C05446=1006.982,330.511,340.600,169.675,53.827,160.488
C05447=1006.976,330.263,340.633,169.667,53.832,160.487
C05448=1006.972,330.016,340.666,169.659,53.837,160.487
C05449=1006.965,329.768,340.699,169.651,53.842,160.486
C05450=1006.960,329.520,340.733,169.643,53.848,160.486
C05451=1006.954,329.273,340.766,169.635,53.853,160.485
C05452=1006.948,329.025,340.799,169.629,53.858,160.485
C05453=1006.942,328.777,340.832,169.620,53.863,160.484
C05454=1006.937,328.530,340.864,169.613,53.869,160.484
C05455=1006.931,328.282,340.897,169.605,53.874,160.483
C05456=1006.926,328.034,340.930,169.597,53.879,160.483
C05457=1006.919,327.786,340.963,169.589,53.885,160.483
C05458=1006.915,327.538,340.995,169.582,53.890,160.482
C05459=1006.909,327.290,341.029,169.575,53.895,160.482
C05460=1006.903,327.043,341.061,169.567,53.900,160.481
C05461=1006.897,326.795,341.095,169.559,53.906,160.481
C05462=1006.893,326.547,341.127,169.552,53.911,160.481
C05463=1006.886,326.300,341.160,169.544,53.916,160.480
C05464=1006.881,326.051,341.192,169.537,53.922,160.480
C05465=1006.876,325.804,341.225,169.529,53.927,160.480
C05466=1006.870,325.556,341.258,169.521,53.932,160.479
C05467=1006.865,325.308,341.290,169.514,53.938,160.479
C05468=1006.859,325.061,341.323,169.507,53.943,160.478
C05469=1006.852,324.704,341.370,169.495,53.951,160.478
C05470=1006.844,324.349,341.417,169.485,53.959,160.477
C05471=1006.835,323.993,341.462,169.474,53.967,160.477
C05472=1006.827,323.638,341.509,169.464,53.974,160.476
C05473=1006.822,323.391,341.540,169.456,53.980,160.476
C05474=1006.816,323.142,341.572,169.449,53.985,160.476
C05475=1006.810,322.895,341.604,169.441,53.990,160.475
C05476=1006.805,322.646,341.637,169.434,53.996,160.475
C05477=1006.800,322.399,341.668,169.426,54.001,160.474
C05478=1006.794,322.151,341.700,169.419,54.007,160.474
C05479=1006.788,321.903,341.732,169.411,54.013,160.474
C05480=1006.782,321.655,341.764,169.404,54.018,160.474
C05481=1006.778,321.407,341.796,169.397,54.024,160.473
C05482=1006.772,321.159,341.828,169.389,54.029,160.473
C05483=1006.766,320.911,341.860,169.382,54.035,160.473
C05484=1006.760,320.663,341.892,169.375,54.040,160.472
C05485=1006.755,320.416,341.924,169.367,54.046,160.472
C05486=1006.749,320.168,341.955,169.360,54.051,160.472
C05487=1006.744,319.920,341.988,169.353,54.057,160.471
C05488=1006.739,319.672,342.020,169.345,54.062,160.471
C05489=1006.733,319.424,342.051,169.338,54.068,160.471
C05490=1006.727,319.176,342.083,169.330,54.074,160.470
C05491=1006.722,318.928,342.114,169.324,54.079,160.470
C05492=1006.717,318.681,342.146,169.316,54.085,160.470
C05493=1006.712,318.432,342.179,169.308,54.090,160.469
C05494=1006.706,318.185,342.210,169.302,54.096,160.469
C05495=1006.701,317.937,342.242,169.294,54.101,160.469
C05496=1006.696,317.689,342.273,169.287,54.108,160.469
C05497=1006.690,317.441,342.305,169.280,54.113,160.468
C05498=1006.685,317.193,342.337,169.273,54.118,160.468
C05499=1006.680,316.945,342.368,169.265,54.124,160.468
C05500=1006.675,316.697,342.400,169.258,54.129,160.467
C05501=1006.669,316.450,342.431,169.251,54.135,160.467
C05502=1006.664,316.202,342.462,169.244,54.141,160.467
C05503=1006.658,315.953,342.494,169.237,54.147,160.467
C05504=1006.654,315.705,342.526,169.229,54.152,160.466
C05505=1006.649,315.457,342.558,169.223,54.158,160.466
C05506=1006.643,315.209,342.589,169.215,54.163,160.466
C05507=1006.638,314.962,342.620,169.208,54.170,160.466
C05508=1006.633,314.714,342.652,169.201,54.175,160.465
C05509=1006.628,314.466,342.683,169.194,54.181,160.465
C05510=1006.623,314.218,342.714,169.187,54.187,160.465
C05511=1006.618,313.970,342.746,169.180,54.192,160.465
C05512=1006.613,313.722,342.777,169.172,54.198,160.464
C05513=1006.607,313.475,342.809,169.166,54.204,160.464
C05514=1006.602,313.226,342.840,169.159,54.210,160.464
C05515=1006.598,312.979,342.872,169.152,54.215,160.464
C05516=1006.593,312.730,342.903,169.145,54.221,160.464
C05517=1006.588,312.482,342.934,169.137,54.227,160.463
C05518=1006.582,312.235,342.965,169.130,54.232,160.463
C05519=1006.577,311.987,342.996,169.123,54.238,160.463
C05520=1006.572,311.739,343.027,169.117,54.244,160.463
C05521=1006.568,311.490,343.059,169.110,54.250,160.462
C05522=1006.562,311.243,343.090,169.102,54.256,160.462
C05523=1006.557,310.994,343.121,169.095,54.261,160.462
C05524=1006.553,310.747,343.152,169.088,54.267,160.462
C05525=1006.548,310.499,343.183,169.082,54.273,160.461
C05526=1006.543,310.251,343.214,169.074,54.279,160.461
C05527=1006.538,310.003,343.246,169.068,54.284,160.461
C05528=1006.533,309.755,343.277,169.061,54.291,160.461
C05529=1006.526,309.405,343.321,169.051,54.299,160.461
C05530=1006.519,309.055,343.365,169.041,54.307,160.460
C05531=1006.512,308.706,343.408,169.032,54.316,160.460
C05532=1006.505,308.356,343.451,169.022,54.324,160.460
C05533=1006.501,308.107,343.483,169.015,54.329,160.460
C05534=1006.496,307.860,343.513,169.008,54.336,160.459
C05535=1006.491,307.612,343.544,169.000,54.341,160.459
C05536=1006.485,307.364,343.574,168.994,54.347,160.459
C05537=1006.481,307.116,343.604,168.987,54.354,160.459
C05538=1006.475,306.868,343.634,168.981,54.359,160.459
C05539=1006.470,306.620,343.665,168.973,54.365,160.458
C05540=1006.465,306.373,343.694,168.967,54.371,160.458
C05541=1006.460,306.124,343.725,168.960,54.377,160.458
C05542=1006.454,305.876,343.755,168.954,54.383,160.458
C05543=1006.449,305.628,343.786,168.946,54.389,160.458
C05544=1006.444,305.380,343.815,168.939,54.396,160.458
C05545=1006.440,305.122,343.847,168.933,54.401,160.458
C05546=1006.434,304.865,343.878,168.926,54.407,160.457
C05547=1006.429,304.606,343.910,168.918,54.414,160.457
C05548=1006.423,304.348,343.941,168.911,54.420,160.457
C05549=1006.180,304.930,343.505,168.907,54.441,160.461
C05550=1006.187,305.298,343.459,168.917,54.432,160.461
C05551=1006.194,305.666,343.415,168.927,54.424,160.461
C05552=1006.203,306.035,343.370,168.937,54.414,160.462
C05553=1006.210,306.403,343.325,168.948,54.405,160.462
C05554=1006.215,306.650,343.295,168.954,54.399,160.462
C05555=1006.220,306.899,343.265,168.962,54.394,160.462
C05556=1006.225,307.147,343.235,168.968,54.388,160.462
C05557=1006.229,307.395,343.205,168.975,54.381,160.463
C05558=1006.235,307.643,343.175,168.982,54.376,160.463
C05559=1006.240,307.891,343.144,168.989,54.370,160.463
C05560=1006.245,308.138,343.113,168.995,54.364,160.463
C05561=1006.250,308.386,343.082,169.003,54.358,160.463
C05562=1006.257,308.739,343.039,169.012,54.350,160.464
C05563=1006.264,309.090,342.995,169.022,54.342,160.464
C05564=1006.270,309.442,342.950,169.032,54.334,160.464
C05565=1006.277,309.795,342.907,169.042,54.326,160.465
C05566=1006.282,310.043,342.876,169.049,54.319,160.465
C05567=1006.287,310.291,342.845,169.056,54.314,160.465
C05568=1006.293,310.539,342.813,169.063,54.308,160.466
C05569=1006.296,310.786,342.782,169.069,54.302,160.465
C05570=1006.301,311.035,342.751,169.077,54.297,160.466
C05571=1006.306,311.283,342.720,169.083,54.291,160.466
C05572=1006.312,311.531,342.689,169.091,54.285,160.466
C05573=1006.317,311.779,342.658,169.097,54.280,160.467
C05574=1006.321,312.027,342.626,169.104,54.273,160.467
C05575=1006.326,312.274,342.596,169.111,54.268,160.467
C05576=1006.331,312.522,342.565,169.119,54.262,160.467
C05577=1006.336,312.770,342.533,169.125,54.256,160.467
C05578=1006.341,313.018,342.502,169.133,54.251,160.468
C05579=1006.346,313.266,342.471,169.140,54.245,160.468
C05580=1006.351,313.514,342.439,169.147,54.240,160.468
C05581=1006.356,313.762,342.408,169.154,54.233,160.468
C05582=1006.361,314.010,342.377,169.161,54.228,160.469
C05583=1006.367,314.258,342.345,169.168,54.222,160.469
C05584=1006.372,314.506,342.314,169.175,54.217,160.469
C05585=1006.377,314.753,342.283,169.182,54.211,160.469
C05586=1006.381,315.002,342.251,169.190,54.205,160.470
C05587=1006.387,315.249,342.219,169.196,54.200,160.470
C05588=1006.392,315.497,342.188,169.204,54.194,160.470
C05589=1006.397,315.745,342.157,169.210,54.189,160.471
C05590=1006.402,315.993,342.126,169.218,54.183,160.471
C05591=1006.408,316.242,342.093,169.225,54.177,160.471
C05592=1006.413,316.490,342.062,169.232,54.172,160.471
C05593=1006.418,316.737,342.031,169.239,54.166,160.472
C05594=1006.423,316.985,342.000,169.247,54.160,160.472
C05595=1006.428,317.233,341.968,169.254,54.155,160.472
C05596=1006.434,317.480,341.936,169.261,54.149,160.473
C05597=1006.439,317.730,341.904,169.268,54.144,160.473
C05598=1006.444,317.977,341.873,169.276,54.138,160.473
C05599=1006.450,318.225,341.841,169.283,54.133,160.474
C05600=1006.455,318.473,341.810,169.290,54.127,160.474
C05601=1006.460,318.720,341.779,169.298,54.122,160.474
C05602=1006.466,318.968,341.747,169.305,54.116,160.475
C05603=1006.471,319.216,341.714,169.312,54.111,160.475
C05604=1006.476,319.464,341.683,169.319,54.105,160.475
C05605=1006.482,319.713,341.651,169.327,54.099,160.476
C05606=1006.487,319.960,341.620,169.334,54.094,160.476
C05607=1006.493,320.208,341.588,169.341,54.088,160.476
C05608=1006.498,320.456,341.555,169.349,54.083,160.477
C05609=1006.503,320.704,341.524,169.356,54.078,160.477
C05610=1006.509,320.951,341.492,169.363,54.072,160.477
C05611=1006.515,321.199,341.460,169.371,54.066,160.478
C05612=1006.520,321.447,341.428,169.378,54.061,160.478
C05613=1006.526,321.695,341.396,169.385,54.055,160.478
C05614=1006.531,321.943,341.364,169.393,54.050,160.478
C05615=1006.536,322.190,341.332,169.401,54.045,160.479
C05616=1006.542,322.439,341.300,169.407,54.039,160.479
C05617=1006.547,322.686,341.269,169.415,54.034,160.480
C05618=1006.553,322.934,341.237,169.423,54.028,160.480
C05619=1006.558,323.182,341.204,169.430,54.022,160.480
C05620=1006.564,323.430,341.172,169.437,54.017,160.481
C05621=1006.569,323.678,341.141,169.445,54.012,160.481
C05622=1006.578,324.036,341.095,169.456,54.004,160.482
C05623=1006.586,324.394,341.048,169.466,53.997,160.482
C05624=1006.594,324.752,341.002,169.478,53.989,160.483
C05625=1006.602,325.110,340.954,169.489,53.981,160.483
C05626=1006.607,325.358,340.922,169.495,53.976,160.484
C05627=1006.613,325.605,340.889,169.503,53.971,160.484
C05628=1006.618,325.854,340.857,169.511,53.965,160.485
C05629=1006.623,326.101,340.824,169.519,53.959,160.485
C05630=1006.629,326.348,340.791,169.526,53.955,160.485
C05631=1006.635,326.597,340.758,169.533,53.949,160.486
C05632=1006.639,326.844,340.725,169.542,53.944,160.486
C05633=1006.645,327.092,340.693,169.549,53.938,160.487
C05634=1006.651,327.340,340.660,169.556,53.933,160.487
C05635=1006.657,327.587,340.628,169.564,53.928,160.487
C05636=1006.662,327.836,340.595,169.572,53.923,160.488
C05637=1006.668,328.084,340.562,169.580,53.918,160.488
C05638=1006.674,328.331,340.529,169.587,53.912,160.489
C05639=1006.679,328.578,340.496,169.594,53.907,160.489
C05640=1006.684,328.827,340.463,169.602,53.902,160.489
C05641=1006.690,329.075,340.430,169.610,53.897,160.490
C05642=1006.696,329.322,340.397,169.618,53.891,160.490
C05643=1006.701,329.570,340.364,169.626,53.886,160.491
C05644=1006.707,329.817,340.331,169.633,53.882,160.491
C05645=1006.713,330.065,340.298,169.641,53.876,160.492
C05646=1006.719,330.313,340.265,169.649,53.871,160.492
C05647=1006.725,330.561,340.232,169.656,53.865,160.493
C05648=1006.730,330.809,340.199,169.664,53.860,160.493
C05649=1006.736,331.056,340.166,169.672,53.856,160.494
C05650=1006.741,331.303,340.133,169.679,53.850,160.494
C05651=1006.747,331.551,340.100,169.687,53.845,160.495
C05652=1006.752,331.799,340.066,169.695,53.840,160.495
C05653=1006.758,332.047,340.033,169.703,53.835,160.496
C05654=1006.764,332.295,340.000,169.711,53.830,160.496
C05655=1006.769,332.542,339.966,169.718,53.825,160.497
C05656=1006.775,332.790,339.932,169.726,53.820,160.497
C05657=1006.780,333.038,339.899,169.734,53.815,160.498
C05658=1006.787,333.286,339.866,169.742,53.809,160.498
C05659=1006.793,333.533,339.832,169.750,53.804,160.499
C05660=1006.798,333.781,339.799,169.758,53.800,160.499
C05661=1006.804,334.029,339.765,169.766,53.795,160.500
C05662=1006.810,334.276,339.731,169.774,53.790,160.500
C05663=1006.815,334.524,339.698,169.782,53.785,160.501
C05664=1006.821,334.771,339.664,169.789,53.779,160.501
C05665=1006.827,335.019,339.631,169.797,53.774,160.502
C05666=1006.833,335.268,339.597,169.805,53.769,160.502
C05667=1006.839,335.515,339.563,169.813,53.765,160.503
C05668=1006.845,335.763,339.530,169.822,53.760,160.503
C05669=1006.851,336.010,339.496,169.830,53.755,160.504
C05670=1006.857,336.257,339.462,169.838,53.750,160.504
C05671=1006.862,336.505,339.429,169.846,53.745,160.505
C05672=1006.869,336.753,339.394,169.854,53.740,160.506
C05673=1006.874,337.001,339.361,169.862,53.735,160.506
C05674=1006.880,337.248,339.327,169.870,53.730,160.507
C05675=1006.886,337.496,339.293,169.877,53.725,160.507
C05676=1006.892,337.744,339.258,169.885,53.720,160.508
C05677=1006.898,337.991,339.225,169.893,53.715,160.508
C05678=1006.904,338.239,339.191,169.902,53.710,160.509
C05679=1006.910,338.486,339.157,169.910,53.706,160.510
C05680=1006.916,338.734,339.123,169.918,53.701,160.510
C05681=1006.921,338.982,339.088,169.926,53.696,160.511
C05682=1006.929,339.306,339.043,169.937,53.689,160.511
C05683=1006.937,339.630,338.999,169.948,53.683,160.512
C05684=1006.945,339.955,338.953,169.958,53.677,160.513
C05685=1006.953,340.279,338.909,169.969,53.671,160.514
C05686=1006.959,340.527,338.874,169.977,53.666,160.515
C05687=1006.964,340.774,338.839,169.985,53.661,160.515
C05688=1006.971,341.022,338.805,169.994,53.656,160.516
C05689=1006.977,341.270,338.771,170.002,53.651,160.516
C05690=1006.983,341.518,338.737,170.010,53.647,160.517
C05691=1006.989,341.765,338.703,170.018,53.642,160.518
C05692=1006.995,342.013,338.667,170.026,53.637,160.518
C05693=1007.001,342.260,338.633,170.035,53.633,160.519
C05694=1007.007,342.508,338.598,170.043,53.628,160.519
C05695=1007.013,342.755,338.564,170.052,53.624,160.520
C05696=1007.020,343.003,338.529,170.060,53.619,160.521
C05697=1007.025,343.250,338.494,170.068,53.614,160.521
C05698=1007.032,343.498,338.459,170.076,53.610,160.522
C05699=1007.038,343.745,338.425,170.085,53.605,160.523
C05700=1007.044,343.993,338.391,170.093,53.600,160.523
C05701=1007.050,344.240,338.355,170.102,53.595,160.524
C05702=1006.736,342.085,338.297,170.011,53.676,160.524
C05703=1006.730,341.839,338.332,170.002,53.680,160.523
C05704=1006.724,341.591,338.366,169.994,53.685,160.523
C05705=1006.718,341.343,338.401,169.986,53.690,160.522
C05706=1006.713,341.096,338.435,169.978,53.695,160.521
C05707=1006.706,340.848,338.470,169.970,53.700,160.521
C05708=1006.700,340.600,338.504,169.961,53.704,160.520
C05709=1006.694,340.353,338.538,169.953,53.709,160.520
C05710=1006.688,340.105,338.572,169.945,53.714,160.519
C05711=1006.682,339.837,338.609,169.936,53.719,160.518
C05712=1006.676,339.568,338.647,169.927,53.725,160.518
C05713=1006.669,339.300,338.685,169.918,53.729,160.517
C05714=1006.663,339.031,338.721,169.909,53.734,160.516
C05715=1006.657,338.784,338.755,169.901,53.739,160.516
C05716=1006.651,338.536,338.789,169.893,53.744,160.515
C05717=1006.645,338.289,338.823,169.885,53.749,160.515
C05718=1006.639,338.041,338.857,169.876,53.754,160.514
C05719=1006.633,337.794,338.891,169.868,53.758,160.513
C05720=1006.628,337.545,338.926,169.860,53.763,160.513
C05721=1006.622,337.298,338.960,169.853,53.768,160.512
C05722=1006.616,337.050,338.994,169.845,53.773,160.512
C05723=1006.610,336.803,339.027,169.837,53.778,160.511
C05724=1006.604,336.556,339.061,169.828,53.783,160.510
C05725=1006.597,336.307,339.094,169.820,53.788,160.510
C05726=1006.592,336.060,339.128,169.812,53.793,160.509
C05727=1006.586,335.812,339.162,169.804,53.798,160.509
C05728=1006.580,335.565,339.196,169.796,53.803,160.508
C05729=1006.575,335.317,339.229,169.788,53.808,160.508
C05730=1006.569,335.069,339.263,169.780,53.813,160.507
C05731=1006.563,334.821,339.297,169.773,53.817,160.507
C05732=1006.557,334.574,339.331,169.765,53.822,160.506
C05733=1006.551,334.327,339.363,169.757,53.827,160.505
C05734=1006.546,334.079,339.397,169.748,53.832,160.505
C05735=1006.540,333.831,339.431,169.740,53.837,160.504
C05736=1006.534,333.583,339.464,169.733,53.843,160.504
C05737=1006.529,333.336,339.497,169.725,53.848,160.503
C05738=1006.523,333.088,339.531,169.716,53.853,160.503
C05739=1006.517,332.840,339.565,169.709,53.857,160.502
C05740=1006.512,332.592,339.598,169.701,53.862,160.502
C05741=1006.506,332.345,339.631,169.693,53.867,160.501
C05742=1006.500,332.097,339.665,169.686,53.873,160.501
C05743=1006.494,331.849,339.698,169.677,53.878,160.500
C05744=1006.489,331.601,339.731,169.670,53.882,160.500
C05745=1006.483,331.354,339.765,169.662,53.887,160.499
C05746=1006.477,331.106,339.798,169.654,53.892,160.499
C05747=1006.472,330.858,339.832,169.646,53.898,160.498
C05748=1006.467,330.611,339.865,169.638,53.903,160.498
C05749=1006.460,330.363,339.897,169.630,53.908,160.497
C05750=1006.455,330.115,339.930,169.624,53.913,160.497
C05751=1006.449,329.867,339.963,169.616,53.918,160.496
C05752=1006.443,329.619,339.996,169.607,53.923,160.496
C05753=1006.438,329.372,340.029,169.600,53.929,160.495
C05754=1006.432,329.124,340.062,169.592,53.934,160.495
C05755=1006.427,328.876,340.094,169.585,53.939,160.495
C05756=1006.421,328.628,340.128,169.577,53.944,160.494
C05757=1006.416,328.381,340.160,169.569,53.949,160.493
C05758=1006.410,328.133,340.193,169.561,53.954,160.493
C05759=1006.405,327.885,340.226,169.554,53.959,160.493
C05760=1006.399,327.638,340.258,169.547,53.965,160.492
C05761=1006.394,327.390,340.292,169.538,53.970,160.492
C05762=1006.388,327.142,340.324,169.531,53.975,160.491
C05763=1006.383,326.894,340.357,169.524,53.980,160.491
C05764=1006.377,326.646,340.389,169.516,53.986,160.491
C05765=1006.371,326.398,340.422,169.508,53.991,160.490
C05766=1006.366,326.151,340.454,169.500,53.996,160.490
C05767=1006.361,325.903,340.488,169.493,54.001,160.489
C05768=1006.355,325.656,340.520,169.486,54.006,160.489
C05769=1006.350,325.407,340.553,169.478,54.012,160.488
C05770=1006.345,325.159,340.585,169.470,54.017,160.488
C05771=1006.337,324.799,340.633,169.460,54.025,160.487
C05772=1006.329,324.439,340.680,169.448,54.033,160.487
C05773=1006.321,324.078,340.726,169.437,54.041,160.486
C05774=1006.312,323.719,340.772,169.427,54.048,160.486
C05775=1006.307,323.470,340.805,169.419,54.053,160.485
C05776=1006.302,323.222,340.837,169.411,54.059,160.485
C05777=1006.296,322.974,340.869,169.405,54.064,160.485
C05778=1006.290,322.727,340.900,169.397,54.070,160.484
C05779=1006.284,322.479,340.932,169.389,54.075,160.484
C05780=1006.280,322.231,340.965,169.381,54.080,160.483
C05781=1006.274,321.983,340.996,169.375,54.086,160.483
C05782=1006.268,321.735,341.028,169.367,54.091,160.483
C05783=1006.263,321.487,341.060,169.360,54.097,160.482
C05784=1006.257,321.239,341.092,169.352,54.102,160.482
C05785=1006.252,320.992,341.124,169.345,54.107,160.481
C05786=1006.247,320.744,341.156,169.337,54.113,160.481
C05787=1006.241,320.496,341.188,169.331,54.118,160.481
C05788=1006.235,320.248,341.220,169.323,54.124,160.480
C05789=1006.230,320.000,341.250,169.315,54.129,160.480
C05790=1006.224,319.752,341.282,169.309,54.135,160.480
C05791=1006.219,319.504,341.314,169.301,54.140,160.479
C05792=1006.214,319.257,341.346,169.293,54.145,160.479
C05793=1006.209,319.009,341.378,169.286,54.151,160.479
C05794=1006.203,318.760,341.409,169.279,54.156,160.478
C05795=1006.198,318.513,341.441,169.271,54.162,160.478
C05796=1006.193,318.265,341.473,169.264,54.167,160.478
C05797=1006.188,318.017,341.504,169.257,54.173,160.477
C05798=1006.183,317.769,341.536,169.250,54.178,160.477
C05799=1006.177,317.521,341.568,169.242,54.184,160.477
C05800=1006.172,317.273,341.599,169.235,54.190,160.476
C05801=1006.166,317.025,341.631,169.228,54.195,160.476
C05802=1006.161,316.777,341.661,169.221,54.201,160.476
C05803=1006.157,316.529,341.694,169.214,54.206,160.475
C05804=1006.152,316.281,341.725,169.206,54.212,160.475
C05805=1006.146,316.034,341.756,169.199,54.218,160.475
C05806=1006.141,315.786,341.787,169.193,54.223,160.475
C05807=1006.136,315.538,341.819,169.185,54.229,160.474
C05808=1006.131,315.290,341.850,169.178,54.234,160.474
C05809=1006.126,315.042,341.882,169.171,54.240,160.474
C05810=1006.121,314.794,341.913,169.163,54.246,160.473
C05811=1006.116,314.546,341.945,169.156,54.251,160.473
C05812=1006.110,314.298,341.976,169.149,54.257,160.473
C05813=1006.105,314.050,342.007,169.143,54.262,160.473
C05814=1006.101,313.802,342.039,169.135,54.268,160.472
C05815=1006.096,313.554,342.070,169.128,54.273,160.472
C05816=1006.091,313.306,342.101,169.121,54.279,160.472
C05817=1006.085,313.059,342.132,169.114,54.284,160.471
C05818=1006.080,312.810,342.163,169.107,54.290,160.471
C05819=1006.075,312.562,342.194,169.100,54.296,160.471
C05820=1006.071,312.314,342.226,169.093,54.302,160.471
C05821=1006.065,312.066,342.258,169.086,54.307,160.470
C05822=1006.061,311.819,342.288,169.079,54.313,160.470
C05823=1006.056,311.571,342.319,169.071,54.319,160.470
C05824=1006.051,311.323,342.350,169.065,54.324,160.470
C05825=1006.046,311.074,342.382,169.057,54.330,160.469
C05826=1006.041,310.826,342.413,169.051,54.336,160.469
C05827=1006.036,310.578,342.443,169.043,54.342,160.469
C05828=1006.031,310.331,342.475,169.037,54.347,160.469
C05829=1006.026,310.083,342.506,169.030,54.353,160.468
C05830=1006.021,309.835,342.537,169.023,54.359,160.468
C05831=1006.015,309.480,342.581,169.013,54.367,160.468
C05832=1006.008,309.126,342.625,169.004,54.375,160.468
C05833=1006.002,308.772,342.669,168.993,54.383,160.467
C05834=1005.994,308.417,342.713,168.984,54.391,160.467
C05835=1005.989,308.169,342.744,168.977,54.398,160.467
C05836=1005.985,307.922,342.775,168.970,54.403,160.466
C05837=1005.980,307.673,342.806,168.963,54.409,160.466
C05838=1005.975,307.426,342.835,168.956,54.415,160.466
C05839=1005.970,307.184,342.865,168.949,54.421,160.466
C05840=1005.965,306.942,342.895,168.942,54.426,160.466
C05841=1005.960,306.700,342.924,168.936,54.432,160.465
C05842=1005.955,306.459,342.953,168.930,54.438,160.465
C05843=1005.950,306.217,342.983,168.922,54.443,160.465
C05844=1005.945,305.976,343.012,168.916,54.449,160.465
C05845=1005.941,305.734,343.041,168.909,54.455,160.465
C05846=1005.935,305.492,343.070,168.902,54.461,160.464
C05847=1005.691,306.038,342.638,168.898,54.480,160.468
C05848=1005.698,306.392,342.595,168.908,54.471,160.468
C05849=1005.705,306.747,342.553,168.918,54.463,160.468
C05850=1005.713,307.102,342.509,168.928,54.454,160.469
C05851=1005.719,307.456,342.466,168.937,54.446,160.469
C05852=1005.725,307.704,342.436,168.944,54.441,160.469
C05853=1005.730,307.952,342.405,168.951,54.434,160.469
C05854=1005.735,308.200,342.374,168.958,54.429,160.470
C05855=1005.739,308.448,342.344,168.965,54.423,160.470
C05856=1005.746,308.805,342.300,168.975,54.415,160.470
C05857=1005.753,309.162,342.256,168.985,54.407,160.471
C05858=1005.760,309.517,342.211,168.994,54.398,160.471
C05859=1005.766,309.874,342.166,169.004,54.390,160.471
C05860=1005.772,310.122,342.135,169.012,54.384,160.472
C05861=1005.777,310.370,342.104,169.018,54.379,160.472
C05862=1005.781,310.619,342.073,169.026,54.373,160.472
C05863=1005.785,310.866,342.042,169.032,54.367,160.472
C05864=1005.790,311.114,342.011,169.040,54.362,160.473
C05865=1005.796,311.362,341.980,169.046,54.356,160.473
C05866=1005.801,311.611,341.949,169.053,54.351,160.473
C05867=1005.805,311.859,341.918,169.061,54.345,160.474
C05868=1005.809,312.106,341.887,169.067,54.339,160.474
C05869=1005.815,312.354,341.856,169.074,54.334,160.474
C05870=1005.820,312.602,341.825,169.081,54.328,160.474
C05871=1005.825,312.850,341.794,169.089,54.323,160.475
C05872=1005.830,313.098,341.763,169.095,54.317,160.475
C05873=1005.834,313.347,341.731,169.103,54.312,160.475
C05874=1005.839,313.594,341.700,169.109,54.306,160.475
C05875=1005.844,313.842,341.669,169.117,54.300,160.476
C05876=1005.849,314.090,341.638,169.124,54.294,160.476
C05877=1005.855,314.337,341.606,169.131,54.289,160.476
C05878=1005.860,314.586,341.575,169.139,54.283,160.477
C05879=1005.864,314.834,341.544,169.145,54.278,160.477
C05880=1005.870,315.081,341.512,169.153,54.272,160.477
C05881=1005.875,315.330,341.481,169.160,54.267,160.478
C05882=1005.880,315.578,341.450,169.167,54.262,160.478
C05883=1005.885,315.825,341.419,169.174,54.256,160.478
C05884=1005.889,316.074,341.387,169.181,54.251,160.479
C05885=1005.895,316.321,341.356,169.188,54.245,160.479
C05886=1005.900,316.569,341.325,169.196,54.240,160.479
C05887=1005.905,316.817,341.293,169.203,54.234,160.480
C05888=1005.911,317.066,341.262,169.210,54.229,160.480
C05889=1005.916,317.313,341.230,169.218,54.223,160.480
C05890=1005.921,317.562,341.198,169.224,54.218,160.480
C05891=1005.926,317.809,341.167,169.232,54.212,160.481
C05892=1005.931,318.057,341.135,169.239,54.206,160.481
C05893=1005.937,318.305,341.104,169.246,54.201,160.481
C05894=1005.942,318.552,341.072,169.254,54.195,160.482
C05895=1005.947,318.801,341.040,169.260,54.190,160.482
C05896=1005.952,319.049,341.009,169.268,54.184,160.482
C05897=1005.958,319.296,340.977,169.276,54.179,160.483
C05898=1005.963,319.544,340.946,169.283,54.174,160.483
C05899=1005.969,319.793,340.914,169.290,54.168,160.484
C05900=1005.974,320.040,340.883,169.297,54.163,160.484
C05901=1005.979,320.288,340.850,169.305,54.157,160.484
C05902=1005.984,320.536,340.819,169.312,54.152,160.485
C05903=1005.990,320.785,340.787,169.319,54.147,160.485
C05904=1005.995,321.032,340.756,169.327,54.141,160.485
C05905=1006.001,321.280,340.724,169.335,54.136,160.486
C05906=1006.006,321.528,340.691,169.341,54.131,160.486
C05907=1006.011,321.776,340.660,169.349,54.126,160.487
C05908=1006.017,322.023,340.628,169.357,54.120,160.487
C05909=1006.023,322.271,340.596,169.364,54.115,160.487
C05910=1006.028,322.519,340.564,169.371,54.109,160.488
C05911=1006.034,322.767,340.532,169.379,54.104,160.488
C05912=1006.039,323.015,340.500,169.386,54.099,160.489
C05913=1006.044,323.262,340.468,169.394,54.093,160.489
C05914=1006.050,323.511,340.436,169.402,54.088,160.489
C05915=1006.055,323.758,340.405,169.409,54.082,160.490
C05916=1006.064,324.121,340.359,169.419,54.075,160.490
C05917=1006.072,324.484,340.311,169.431,54.067,160.491
C05918=1006.080,324.846,340.263,169.442,54.059,160.492
C05919=1006.087,325.209,340.216,169.452,54.052,160.492
C05920=1006.093,325.457,340.184,169.460,54.046,160.493
C05921=1006.098,325.705,340.151,169.468,54.041,160.493
C05922=1006.104,325.953,340.118,169.476,54.036,160.494
C05923=1006.109,326.200,340.086,169.483,54.031,160.494
C05924=1006.114,326.448,340.053,169.491,54.025,160.494
C05925=1006.119,326.696,340.021,169.499,54.020,160.495
C05926=1006.125,326.943,339.988,169.505,54.015,160.495
C05927=1006.131,327.192,339.955,169.513,54.010,160.496
C05928=1006.136,327.439,339.923,169.521,54.005,160.496
C05929=1006.142,327.687,339.890,169.529,54.000,160.497
C05930=1006.147,327.935,339.857,169.536,53.995,160.497
C05931=1006.153,328.182,339.825,169.544,53.989,160.498
C05932=1006.158,328.431,339.792,169.552,53.984,160.498
C05933=1006.164,328.679,339.759,169.560,53.979,160.498
C05934=1006.169,328.925,339.726,169.567,53.974,160.499
C05935=1006.175,329.173,339.693,169.575,53.969,160.500
C05936=1006.180,329.422,339.660,169.582,53.963,160.500
C05937=1006.186,329.670,339.628,169.591,53.958,160.500
C05938=1006.191,329.917,339.595,169.598,53.954,160.501
C05939=1006.198,330.164,339.562,169.606,53.949,160.502
C05940=1006.203,330.412,339.528,169.613,53.943,160.502
C05941=1006.208,330.661,339.496,169.622,53.938,160.502
C05942=1006.214,330.908,339.463,169.630,53.933,160.503
C05943=1006.220,331.156,339.430,169.637,53.929,160.504
C05944=1006.225,331.403,339.397,169.644,53.923,160.504
C05945=1006.231,331.651,339.363,169.652,53.918,160.504
C05946=1006.237,331.899,339.329,169.661,53.913,160.505
C05947=1006.242,332.147,339.296,169.669,53.908,160.506
C05948=1006.248,332.394,339.263,169.676,53.904,160.506
C05949=1006.253,332.642,339.230,169.684,53.899,160.507
C05950=1006.258,332.890,339.196,169.691,53.893,160.507
C05951=1006.265,333.137,339.164,169.700,53.888,160.508
C05952=1006.270,333.385,339.130,169.708,53.883,160.508
C05953=1006.276,333.632,339.096,169.715,53.878,160.509
C05954=1006.282,333.880,339.063,169.723,53.873,160.509
C05955=1006.287,334.128,339.030,169.731,53.868,160.510
C05956=1006.293,334.375,338.996,169.739,53.863,160.510
C05957=1006.299,334.623,338.962,169.747,53.858,160.511
C05958=1006.304,334.871,338.929,169.755,53.854,160.512
C05959=1006.310,335.119,338.895,169.763,53.849,160.512
C05960=1006.316,335.366,338.862,169.771,53.844,160.513
C05961=1006.322,335.614,338.829,169.779,53.839,160.513
C05962=1006.328,335.862,338.794,169.787,53.834,160.514
C05963=1006.334,336.110,338.761,169.795,53.829,160.514
C05964=1006.340,336.357,338.727,169.803,53.824,160.515
C05965=1006.345,336.605,338.694,169.811,53.819,160.515
C05966=1006.351,336.852,338.660,169.819,53.814,160.516
C05967=1006.357,337.100,338.626,169.828,53.810,160.517
C05968=1006.362,337.348,338.592,169.836,53.805,160.517
C05969=1006.369,337.596,338.558,169.844,53.800,160.518
C05970=1006.375,337.843,338.524,169.851,53.795,160.518
C05971=1006.380,338.091,338.490,169.859,53.790,160.519
C05972=1006.386,338.338,338.456,169.867,53.785,160.520
C05973=1006.392,338.585,338.422,169.876,53.781,160.520
C05974=1006.398,338.834,338.389,169.884,53.776,160.521
C05975=1006.403,339.082,338.354,169.892,53.771,160.521
C05976=1006.409,339.293,338.325,169.900,53.767,160.522
C05977=1006.413,339.505,338.296,169.906,53.763,160.522
C05978=1006.419,339.717,338.266,169.913,53.759,160.523
C05979=1006.424,339.930,338.237,169.920,53.755,160.524
C05980=1006.113,337.770,338.173,169.831,53.833,160.523
C05981=1006.107,337.523,338.207,169.823,53.838,160.522
C05982=1006.102,337.275,338.242,169.814,53.842,160.522
C05983=1006.096,337.027,338.275,169.806,53.847,160.521
C05984=1006.090,336.779,338.310,169.799,53.852,160.521
C05985=1006.084,336.532,338.342,169.791,53.857,160.520
C05986=1006.078,336.284,338.376,169.783,53.862,160.519
C05987=1006.072,336.036,338.410,169.774,53.867,160.519
C05988=1006.067,335.789,338.443,169.766,53.872,160.518
C05989=1006.061,335.541,338.477,169.758,53.876,160.517
C05990=1006.056,335.293,338.510,169.750,53.881,160.517
C05991=1006.050,335.046,338.544,169.742,53.886,160.516
C05992=1006.044,334.798,338.578,169.734,53.890,160.516
C05993=1006.039,334.550,338.611,169.726,53.895,160.515
C05994=1006.032,334.303,338.644,169.718,53.900,160.515
C05995=1006.026,334.055,338.678,169.710,53.905,160.514
C05996=1006.021,333.808,338.711,169.702,53.910,160.513
C05997=1006.015,333.560,338.745,169.694,53.915,160.513
C05998=1006.010,333.312,338.778,169.687,53.920,160.512
C05999=1006.004,333.064,338.811,169.679,53.925,160.512
C06000=1005.998,332.817,338.845,169.671,53.930,160.511
C06001=1005.993,332.569,338.879,169.662,53.935,160.511
C06002=1005.987,332.321,338.912,169.654,53.940,160.510
C06003=1005.981,332.074,338.944,169.648,53.945,160.510
C06004=1005.976,331.826,338.978,169.640,53.950,160.509
C06005=1005.970,331.578,339.011,169.632,53.955,160.509
C06006=1005.965,331.330,339.044,169.623,53.960,160.508
C06007=1005.959,331.082,339.078,169.616,53.965,160.508
C06008=1005.954,330.834,339.111,169.608,53.970,160.507
C06009=1005.949,330.587,339.144,169.600,53.975,160.506
C06010=1005.942,330.339,339.177,169.592,53.980,160.506
C06011=1005.937,330.091,339.209,169.584,53.985,160.506
C06012=1005.932,329.844,339.242,169.577,53.990,160.505
C06013=1005.926,329.596,339.275,169.569,53.995,160.504
C06014=1005.920,329.348,339.308,169.562,54.001,160.504
C06015=1005.914,329.100,339.340,169.553,54.006,160.504
C06016=1005.909,328.853,339.373,169.546,54.010,160.503
C06017=1005.904,328.605,339.407,169.538,54.015,160.502
C06018=1005.898,328.357,339.439,169.531,54.021,160.502
C06019=1005.893,328.110,339.472,169.523,54.025,160.502
C06020=1005.887,327.862,339.505,169.515,54.030,160.501
C06021=1005.881,327.613,339.537,169.508,54.036,160.501
C06022=1005.877,327.366,339.570,169.500,54.041,160.500
C06023=1005.871,327.118,339.602,169.493,54.046,160.500
C06024=1005.866,326.871,339.635,169.485,54.051,160.499
C06025=1005.860,326.622,339.668,169.477,54.056,160.499
C06026=1005.854,326.375,339.700,169.470,54.061,160.498
C06027=1005.849,326.127,339.733,169.462,54.066,160.498
C06028=1005.844,325.879,339.766,169.454,54.072,160.497
C06029=1005.838,325.631,339.798,169.447,54.077,160.497
C06030=1005.833,325.383,339.830,169.439,54.082,160.496
C06031=1005.828,325.136,339.863,169.432,54.087,160.496
C06032=1005.822,324.887,339.895,169.423,54.092,160.495
C06033=1005.817,324.616,339.931,169.416,54.098,160.495
C06034=1005.811,324.343,339.967,169.407,54.104,160.495
C06035=1005.804,324.071,340.002,169.400,54.110,160.494
C06036=1005.798,323.799,340.036,169.391,54.116,160.494
C06037=1005.794,323.551,340.069,169.384,54.120,160.493
C06038=1005.788,323.303,340.101,169.376,54.126,160.493
C06039=1005.782,323.055,340.132,169.368,54.131,160.492
C06040=1005.776,322.807,340.164,169.361,54.136,160.492
C06041=1005.771,322.559,340.196,169.354,54.142,160.492
C06042=1005.766,322.312,340.228,169.346,54.147,160.491
C06043=1005.760,322.063,340.260,169.339,54.152,160.491
C06044=1005.755,321.816,340.292,169.331,54.158,160.490
C06045=1005.750,321.568,340.323,169.323,54.163,160.490
C06046=1005.744,321.319,340.355,169.317,54.168,160.490
C06047=1005.738,321.072,340.387,169.309,54.174,160.489
C06048=1005.734,320.824,340.419,169.302,54.179,160.489
C06049=1005.728,320.576,340.451,169.294,54.184,160.488
C06050=1005.723,320.328,340.482,169.287,54.190,160.488
C06051=1005.717,320.080,340.513,169.280,54.195,160.488
C06052=1005.712,319.833,340.545,169.272,54.200,160.487
C06053=1005.706,319.585,340.577,169.264,54.206,160.487
C06054=1005.702,319.336,340.609,169.258,54.211,160.486
C06055=1005.696,319.089,340.640,169.250,54.217,160.486
C06056=1005.691,318.841,340.672,169.243,54.222,160.486
C06057=1005.686,318.593,340.703,169.235,54.227,160.485
C06058=1005.680,318.345,340.735,169.229,54.232,160.485
C06059=1005.675,318.096,340.767,169.221,54.238,160.485
C06060=1005.670,317.849,340.798,169.213,54.244,160.484
C06061=1005.665,317.601,340.829,169.207,54.249,160.484
C06062=1005.660,317.353,340.861,169.199,54.255,160.484
C06063=1005.655,317.105,340.892,169.193,54.260,160.483
C06064=1005.649,316.858,340.923,169.185,54.266,160.483
C06065=1005.645,316.609,340.955,169.178,54.270,160.482
C06066=1005.639,316.362,340.987,169.170,54.276,160.482
C06067=1005.634,316.113,341.018,169.164,54.281,160.482
C06068=1005.629,315.866,341.049,169.156,54.287,160.481
C06069=1005.624,315.618,341.080,169.148,54.293,160.481
C06070=1005.620,315.369,341.112,169.142,54.298,160.481
C06071=1005.614,315.122,341.143,169.134,54.304,160.480
C06072=1005.609,314.874,341.174,169.127,54.309,160.480
C06073=1005.604,314.626,341.205,169.120,54.315,160.480
C06074=1005.599,314.378,341.237,169.113,54.320,160.479
C06075=1005.594,314.130,341.268,169.106,54.326,160.479
C06076=1005.589,313.881,341.299,169.099,54.331,160.479
C06077=1005.584,313.634,341.331,169.091,54.337,160.478
C06078=1005.579,313.387,341.362,169.085,54.342,160.478
C06079=1005.574,313.138,341.393,169.077,54.348,160.478
C06080=1005.569,312.890,341.424,169.070,54.353,160.478
C06081=1005.565,312.642,341.455,169.063,54.359,160.477
C06082=1005.560,312.394,341.486,169.057,54.365,160.477
C06083=1005.554,312.146,341.518,169.050,54.370,160.477
C06084=1005.550,311.899,341.548,169.042,54.376,160.476
C06085=1005.545,311.651,341.579,169.036,54.381,160.476
C06086=1005.540,311.402,341.610,169.028,54.387,160.476
C06087=1005.535,311.154,341.642,169.022,54.392,160.476
C06088=1005.531,310.907,341.672,169.014,54.398,160.475
C06089=1005.526,310.658,341.703,169.008,54.404,160.475
C06090=1005.521,310.410,341.734,169.000,54.409,160.475
C06091=1005.516,310.162,341.765,168.993,54.415,160.474
C06092=1005.512,309.914,341.796,168.986,54.420,160.474
C06093=1005.504,309.556,341.841,168.976,54.429,160.474
C06094=1005.498,309.197,341.885,168.966,54.437,160.473
C06095=1005.491,308.837,341.930,168.956,54.445,160.473
C06096=1005.484,308.479,341.975,168.947,54.453,160.473
C06097=1005.480,308.239,342.005,168.940,54.458,160.472
C06098=1005.475,308.000,342.034,168.933,54.464,160.472
C06099=1005.471,307.762,342.063,168.926,54.470,160.472
C06100=1005.465,307.522,342.092,168.920,54.475,160.472
C06101=1005.461,307.284,342.122,168.913,54.481,160.471
C06102=1005.456,307.045,342.151,168.906,54.486,160.471
C06103=1005.452,306.806,342.179,168.900,54.491,160.471
C06104=1005.447,306.567,342.209,168.894,54.497,160.471
C06105=1005.202,307.081,341.780,168.889,54.514,160.474
C06106=1005.209,307.438,341.737,168.899,54.506,160.474
C06107=1005.217,307.795,341.694,168.908,54.497,160.474
C06108=1005.223,308.152,341.650,168.919,54.490,160.475
C06109=1005.229,308.509,341.605,168.928,54.482,160.475
C06110=1005.236,308.870,341.561,168.938,54.473,160.475
C06111=1005.243,309.231,341.515,168.948,54.466,160.476
C06112=1005.250,309.593,341.470,168.959,54.457,160.476
C06113=1005.256,309.954,341.425,168.969,54.449,160.477
C06114=1005.261,310.203,341.395,168.975,54.443,160.477
C06115=1005.266,310.451,341.364,168.983,54.438,160.477
C06116=1005.271,310.698,341.334,168.989,54.432,160.478
C06117=1005.276,310.946,341.303,168.996,54.427,160.478
C06118=1005.280,311.195,341.271,169.004,54.421,160.478
C06119=1005.285,311.442,341.240,169.010,54.416,160.479
C06120=1005.290,311.690,341.210,169.018,54.410,160.479
C06121=1005.295,311.938,341.179,169.025,54.405,160.479
C06122=1005.300,312.186,341.147,169.032,54.399,160.480
C06123=1005.304,312.434,341.116,169.039,54.394,160.480
C06124=1005.309,312.682,341.085,169.045,54.389,160.480
C06125=1005.314,312.930,341.054,169.053,54.383,160.481
C06126=1005.319,313.178,341.023,169.060,54.378,160.481
C06127=1005.324,313.426,340.992,169.067,54.372,160.481
C06128=1005.329,313.674,340.961,169.074,54.367,160.481
C06129=1005.333,313.922,340.929,169.082,54.361,160.482
C06130=1005.338,314.170,340.898,169.088,54.356,160.482
C06131=1005.344,314.418,340.867,169.096,54.350,160.483
C06132=1005.349,314.666,340.836,169.103,54.345,160.483
C06133=1005.354,314.913,340.805,169.110,54.339,160.483
C06134=1005.358,315.162,340.773,169.117,54.334,160.483
C06135=1005.363,315.410,340.742,169.124,54.328,160.484
C06136=1005.369,315.658,340.711,169.131,54.323,160.484
C06137=1005.374,315.906,340.680,169.139,54.317,160.484
C06138=1005.379,316.154,340.649,169.145,54.312,160.485
C06139=1005.384,316.401,340.617,169.153,54.306,160.485
C06140=1005.389,316.650,340.585,169.160,54.301,160.486
C06141=1005.394,316.898,340.554,169.168,54.296,160.486
C06142=1005.399,317.145,340.523,169.174,54.290,160.486
C06143=1005.404,317.394,340.492,169.182,54.285,160.487
C06144=1005.410,317.641,340.460,169.189,54.279,160.487
C06145=1005.414,317.889,340.429,169.196,54.274,160.487
C06146=1005.419,318.137,340.397,169.203,54.269,160.488
C06147=1005.424,318.385,340.366,169.211,54.263,160.488
C06148=1005.430,318.633,340.334,169.219,54.258,160.489
C06149=1005.435,318.880,340.303,169.225,54.252,160.489
C06150=1005.441,319.129,340.271,169.233,54.247,160.489
C06151=1005.446,319.377,340.239,169.240,54.242,160.490
C06152=1005.451,319.625,340.208,169.248,54.236,160.490
C06153=1005.456,319.872,340.177,169.254,54.231,160.490
C06154=1005.461,320.120,340.145,169.262,54.226,160.491
C06155=1005.467,320.369,340.114,169.270,54.220,160.491
C06156=1005.472,320.617,340.081,169.277,54.215,160.492
C06157=1005.477,320.864,340.050,169.285,54.210,160.492
C06158=1005.482,321.112,340.018,169.291,54.205,160.492
C06159=1005.488,321.360,339.987,169.299,54.199,160.493
C06160=1005.494,321.608,339.955,169.307,54.194,160.493
C06161=1005.499,321.855,339.923,169.314,54.189,160.494
C06162=1005.504,322.103,339.891,169.322,54.184,160.494
C06163=1005.510,322.352,339.859,169.328,54.179,160.495
C06164=1005.515,322.600,339.828,169.336,54.173,160.495
C06165=1005.521,322.848,339.796,169.344,54.168,160.496
C06166=1005.526,323.095,339.764,169.351,54.163,160.496
C06167=1005.531,323.343,339.732,169.359,54.158,160.496
C06168=1005.537,323.591,339.700,169.367,54.152,160.497
C06169=1005.542,323.839,339.669,169.374,54.147,160.497
C06170=1005.547,324.070,339.638,169.380,54.142,160.497
C06171=1005.553,324.302,339.609,169.387,54.137,160.498
C06172=1005.558,324.534,339.579,169.395,54.132,160.499
C06173=1005.563,324.766,339.548,169.402,54.127,160.499
C06174=1005.567,324.996,339.518,169.409,54.123,160.499
C06175=1005.572,325.228,339.488,169.416,54.118,160.500
C06176=1005.577,325.459,339.458,169.423,54.113,160.500
C06177=1005.582,325.692,339.427,169.430,54.108,160.501
C06178=1005.588,325.939,339.395,169.438,54.103,160.501
C06179=1005.593,326.187,339.362,169.445,54.099,160.502
C06180=1005.598,326.435,339.329,169.453,54.093,160.502
C06181=1005.604,326.683,339.298,169.461,54.088,160.503
C06182=1005.609,326.931,339.265,169.468,54.083,160.503
C06183=1005.614,327.178,339.232,169.476,54.078,160.503
C06184=1005.620,327.427,339.200,169.484,54.073,160.504
C06185=1005.625,327.674,339.167,169.491,54.068,160.505
C06186=1005.630,327.922,339.134,169.499,54.062,160.505
C06187=1005.636,328.170,339.102,169.507,54.057,160.506
C06188=1005.641,328.417,339.069,169.514,54.053,160.506
C06189=1005.647,328.665,339.037,169.522,54.048,160.507
C06190=1005.653,328.913,339.003,169.530,54.042,160.507
C06191=1005.658,329.161,338.971,169.538,54.037,160.508
C06192=1005.664,329.409,338.938,169.545,54.033,160.508
C06193=1005.669,329.657,338.905,169.553,54.028,160.509
C06194=1005.674,329.904,338.873,169.560,54.022,160.509
C06195=1005.680,330.152,338.840,169.569,54.017,160.510
C06196=1005.686,330.400,338.807,169.576,54.012,160.510
C06197=1005.691,330.648,338.773,169.584,54.007,160.511
C06198=1005.697,330.895,338.741,169.592,54.002,160.511
C06199=1005.703,331.143,338.707,169.600,53.997,160.512
C06200=1005.708,331.391,338.675,169.607,53.993,160.512
C06201=1005.713,331.639,338.642,169.615,53.988,160.513
C06202=1005.719,331.887,338.608,169.623,53.983,160.514
C06203=1005.724,332.134,338.575,169.631,53.978,160.514
C06204=1005.730,332.381,338.541,169.638,53.973,160.514
C06205=1005.735,332.629,338.508,169.646,53.968,160.515
C06206=1005.741,332.877,338.474,169.654,53.963,160.515
C06207=1005.747,333.125,338.442,169.662,53.958,160.516
C06208=1005.753,333.373,338.408,169.669,53.953,160.517
C06209=1005.758,333.621,338.375,169.678,53.949,160.517
C06210=1005.763,333.868,338.342,169.686,53.944,160.518
C06211=1005.769,334.116,338.309,169.694,53.939,160.519
C06212=1005.775,334.363,338.275,169.702,53.934,160.519
C06213=1005.780,334.611,338.241,169.709,53.929,160.520
C06214=1005.786,334.859,338.208,169.718,53.924,160.520
C06215=1005.791,335.107,338.175,169.726,53.919,160.521
C06216=1005.798,335.354,338.141,169.734,53.914,160.521
C06217=1005.804,335.602,338.108,169.742,53.909,160.522
C06218=1005.495,333.430,338.039,169.654,53.985,160.521
C06219=1005.490,333.182,338.072,169.646,53.990,160.520
C06220=1005.484,332.934,338.106,169.638,53.994,160.520
C06221=1005.478,332.687,338.139,169.630,53.999,160.519
C06222=1005.472,332.439,338.172,169.622,54.004,160.518
C06223=1005.468,332.191,338.205,169.614,54.009,160.518
C06224=1005.462,331.944,338.238,169.607,54.014,160.517
C06225=1005.456,331.696,338.272,169.599,54.019,160.517
C06226=1005.451,331.448,338.305,169.591,54.024,160.516
C06227=1005.446,331.201,338.338,169.583,54.029,160.515
C06228=1005.440,330.953,338.371,169.576,54.033,160.515
C06229=1005.435,330.705,338.405,169.568,54.038,160.514
C06230=1005.429,330.457,338.437,169.559,54.043,160.514
C06231=1005.424,330.209,338.470,169.551,54.048,160.513
C06232=1005.418,329.961,338.503,169.544,54.053,160.513
C06233=1005.412,329.714,338.536,169.537,54.058,160.512
C06234=1005.407,329.466,338.568,169.528,54.063,160.512
C06235=1005.401,329.218,338.601,169.521,54.068,160.511
C06236=1005.396,328.970,338.633,169.513,54.073,160.511
C06237=1005.391,328.723,338.666,169.505,54.078,160.510
C06238=1005.385,328.475,338.699,169.497,54.083,160.509
C06239=1005.379,328.227,338.732,169.490,54.088,160.509
C06240=1005.374,327.979,338.765,169.482,54.093,160.509
C06241=1005.368,327.731,338.797,169.474,54.098,160.508
C06242=1005.363,327.484,338.830,169.467,54.103,160.508
C06243=1005.358,327.235,338.862,169.459,54.108,160.507
C06244=1005.353,326.989,338.895,169.451,54.114,160.507
C06245=1005.347,326.740,338.927,169.444,54.118,160.506
C06246=1005.342,326.493,338.959,169.436,54.123,160.505
C06247=1005.336,326.245,338.992,169.428,54.129,160.505
C06248=1005.332,325.997,339.024,169.421,54.133,160.505
C06249=1005.326,325.749,339.056,169.413,54.138,160.504
C06250=1005.321,325.501,339.089,169.407,54.144,160.504
C06251=1005.312,325.096,339.142,169.393,54.152,160.503
C06252=1005.303,324.690,339.195,169.381,54.160,160.502
C06253=1005.294,324.285,339.248,169.369,54.169,160.501
C06254=1005.286,323.879,339.300,169.356,54.177,160.500
C06255=1005.281,323.631,339.332,169.350,54.182,160.500
C06256=1005.275,323.383,339.364,169.342,54.187,160.500
C06257=1005.269,323.135,339.395,169.334,54.193,160.499
C06258=1005.265,322.888,339.428,169.327,54.198,160.499
C06259=1005.259,322.639,339.460,169.319,54.203,160.498
C06260=1005.253,322.392,339.491,169.311,54.208,160.498
C06261=1005.248,322.144,339.523,169.305,54.214,160.497
C06262=1005.243,321.896,339.554,169.296,54.219,160.497
C06263=1005.238,321.648,339.586,169.290,54.224,160.497
C06264=1005.232,321.400,339.618,169.282,54.229,160.496
C06265=1005.227,321.153,339.650,169.274,54.235,160.496
C06266=1005.221,320.904,339.681,169.267,54.240,160.495
C06267=1005.216,320.656,339.713,169.259,54.245,160.495
C06268=1005.210,320.409,339.744,169.253,54.250,160.494
C06269=1005.206,320.160,339.776,169.245,54.255,160.494
C06270=1005.201,319.913,339.808,169.238,54.260,160.494
C06271=1005.195,319.665,339.839,169.230,54.266,160.493
C06272=1005.190,319.416,339.871,169.223,54.271,160.493
C06273=1005.184,319.169,339.902,169.216,54.276,160.492
C06274=1005.180,318.920,339.934,169.208,54.282,160.492
C06275=1005.174,318.673,339.965,169.201,54.287,160.491
C06276=1005.169,318.425,339.996,169.193,54.292,160.491
C06277=1005.164,318.177,340.028,169.187,54.298,160.491
C06278=1005.159,317.929,340.059,169.178,54.303,160.490
C06279=1005.154,317.682,340.091,169.172,54.308,160.490
C06280=1005.149,317.433,340.122,169.164,54.314,160.489
C06281=1005.144,317.186,340.154,169.158,54.319,160.489
C06282=1005.139,316.938,340.185,169.149,54.324,160.489
C06283=1005.133,316.663,340.219,169.142,54.330,160.488
C06284=1005.127,316.389,340.254,169.135,54.336,160.488
C06285=1005.122,316.115,340.289,169.126,54.342,160.488
C06286=1005.116,315.841,340.323,169.118,54.348,160.487
C06287=1005.111,315.593,340.354,169.111,54.354,160.487
C06288=1005.106,315.345,340.385,169.104,54.358,160.486
C06289=1005.101,315.097,340.418,169.096,54.364,160.486
C06290=1005.096,314.849,340.449,169.089,54.369,160.486
C06291=1005.092,314.601,340.479,169.082,54.375,160.485
C06292=1005.087,314.353,340.510,169.075,54.380,160.485
C06293=1005.081,314.106,340.542,169.068,54.386,160.485
C06294=1005.077,313.857,340.573,169.061,54.391,160.484
C06295=1005.072,313.609,340.604,169.054,54.397,160.484
C06296=1005.067,313.361,340.635,169.047,54.402,160.484
C06297=1005.062,313.113,340.666,169.039,54.407,160.483
C06298=1005.057,312.865,340.697,169.032,54.413,160.483
C06299=1005.053,312.617,340.728,169.025,54.418,160.482
C06300=1005.048,312.369,340.759,169.019,54.423,160.482
C06301=1005.043,312.121,340.790,169.011,54.429,160.482
C06302=1005.038,311.873,340.821,169.004,54.434,160.481
C06303=1005.033,311.625,340.852,168.997,54.440,160.481
C06304=1005.028,311.377,340.883,168.990,54.445,160.481
C06305=1005.024,311.129,340.914,168.983,54.451,160.480
C06306=1005.019,310.881,340.945,168.976,54.456,160.480
C06307=1005.014,310.633,340.976,168.969,54.462,160.480
C06308=1005.010,310.386,341.006,168.962,54.467,160.479
C06309=1005.005,310.137,341.037,168.955,54.473,160.479
C06310=1005.001,309.890,341.068,168.949,54.479,160.479
C06311=1004.994,309.552,341.110,168.939,54.486,160.479
C06312=1004.988,309.214,341.152,168.929,54.494,160.478
C06313=1004.981,308.876,341.194,168.920,54.501,160.478
C06314=1004.975,308.539,341.236,168.910,54.508,160.477
C06315=1004.971,308.300,341.266,168.903,54.514,160.477
C06316=1004.966,308.060,341.295,168.897,54.520,160.477
C06317=1004.962,307.821,341.325,168.891,54.525,160.477
C06318=1004.957,307.581,341.354,168.884,54.530,160.476
C06319=1004.711,308.068,340.929,168.880,54.545,160.479
C06320=1004.716,308.319,340.898,168.886,54.540,160.479
C06321=1004.720,308.570,340.866,168.893,54.535,160.479
C06322=1004.727,308.936,340.821,168.903,54.526,160.480
C06323=1004.734,309.302,340.776,168.914,54.518,160.480
C06324=1004.741,309.668,340.730,168.923,54.510,160.481
C06325=1004.748,310.034,340.685,168.935,54.502,160.481
C06326=1004.753,310.282,340.654,168.941,54.497,160.482
C06327=1004.757,310.530,340.623,168.948,54.491,160.482
C06328=1004.762,310.778,340.592,168.955,54.486,160.482
C06329=1004.766,311.026,340.562,168.962,54.480,160.483
C06330=1004.771,311.274,340.531,168.969,54.475,160.483
C06331=1004.776,311.522,340.500,168.976,54.469,160.483
C06332=1004.780,311.770,340.469,168.983,54.464,160.483
C06333=1004.786,312.018,340.438,168.990,54.459,160.484
C06334=1004.791,312.266,340.407,168.997,54.453,160.484
C06335=1004.794,312.514,340.376,169.004,54.448,160.484
C06336=1004.799,312.762,340.345,169.011,54.442,160.485
C06337=1004.805,313.010,340.314,169.018,54.437,160.485
C06338=1004.810,313.258,340.283,169.025,54.432,160.486
C06339=1004.814,313.505,340.252,169.033,54.426,160.486
C06340=1004.819,313.754,340.220,169.039,54.421,160.486
C06341=1004.824,314.002,340.189,169.047,54.415,160.487
C06342=1004.829,314.250,340.159,169.054,54.410,160.487
C06343=1004.834,314.498,340.128,169.060,54.405,160.487
C06344=1004.839,314.746,340.097,169.069,54.400,160.488
C06345=1004.843,314.994,340.065,169.075,54.394,160.488
C06346=1004.848,315.241,340.034,169.083,54.389,160.489
C06347=1004.853,315.489,340.003,169.089,54.383,160.489
C06348=1004.858,315.738,339.972,169.097,54.378,160.489
C06349=1004.863,315.986,339.941,169.104,54.373,160.490
C06350=1004.869,316.233,339.909,169.111,54.368,160.490
C06351=1004.873,316.482,339.878,169.118,54.362,160.490
C06352=1004.878,316.730,339.847,169.125,54.357,160.491
C06353=1004.884,316.977,339.815,169.133,54.352,160.491
C06354=1004.889,317.225,339.784,169.140,54.346,160.492
C06355=1004.894,317.474,339.753,169.147,54.341,160.492
C06356=1004.898,317.721,339.721,169.155,54.336,160.493
C06357=1004.904,317.970,339.690,169.162,54.330,160.493
C06358=1004.909,318.217,339.658,169.169,54.325,160.493
C06359=1004.914,318.465,339.627,169.177,54.320,160.494
C06360=1004.919,318.713,339.596,169.184,54.315,160.494
C06361=1004.924,318.961,339.564,169.191,54.309,160.494
C06362=1004.929,319.209,339.533,169.198,54.305,160.495
C06363=1004.934,319.457,339.502,169.206,54.299,160.495
C06364=1004.940,319.704,339.470,169.213,54.294,160.496
C06365=1004.945,319.952,339.439,169.221,54.289,160.496
C06366=1004.951,320.201,339.407,169.228,54.284,160.497
C06367=1004.955,320.449,339.375,169.235,54.278,160.497
C06368=1004.960,320.697,339.344,169.242,54.273,160.497
C06369=1004.966,320.944,339.312,169.250,54.268,160.498
C06370=1004.971,321.192,339.281,169.258,54.262,160.498
C06371=1004.977,321.440,339.249,169.265,54.258,160.499
C06372=1004.981,321.688,339.217,169.273,54.252,160.499
C06373=1004.987,321.936,339.185,169.280,54.247,160.500
C06374=1004.992,322.184,339.154,169.287,54.242,160.500
C06375=1004.998,322.432,339.122,169.294,54.237,160.501
C06376=1005.003,322.680,339.091,169.302,54.231,160.501
C06377=1005.009,322.927,339.059,169.310,54.226,160.502
C06378=1005.013,323.176,339.027,169.317,54.222,160.502
C06379=1005.019,323.424,338.995,169.325,54.216,160.503
C06380=1005.024,323.671,338.964,169.332,54.211,160.503
C06381=1005.030,323.920,338.932,169.340,54.206,160.503
C06382=1005.037,324.267,338.887,169.350,54.199,160.504
C06383=1005.045,324.615,338.842,169.361,54.192,160.505
C06384=1005.052,324.963,338.796,169.372,54.185,160.506
C06385=1005.060,325.311,338.751,169.382,54.177,160.506
C06386=1005.065,325.558,338.718,169.390,54.172,160.507
C06387=1005.071,325.806,338.686,169.397,54.168,160.507
C06388=1005.075,326.054,338.654,169.405,54.162,160.508
C06389=1005.080,326.303,338.621,169.413,54.157,160.508
C06390=1005.086,326.550,338.589,169.420,54.152,160.509
C06391=1005.091,326.797,338.557,169.428,54.147,160.509
C06392=1005.096,327.045,338.523,169.436,54.142,160.510
C06393=1005.102,327.293,338.492,169.443,54.137,160.510
C06394=1005.107,327.541,338.459,169.451,54.132,160.511
C06395=1005.113,327.789,338.426,169.459,54.127,160.511
C06396=1005.118,328.037,338.394,169.466,54.123,160.512
C06397=1005.123,328.285,338.361,169.474,54.118,160.513
C06398=1005.129,328.532,338.329,169.481,54.113,160.513
C06399=1005.134,328.780,338.296,169.489,54.107,160.513
C06400=1005.139,329.028,338.264,169.497,54.102,160.514
C06401=1005.145,329.276,338.231,169.505,54.097,160.515
C06402=1005.151,329.524,338.198,169.512,54.093,160.515
C06403=1005.156,329.771,338.165,169.520,54.088,160.516
C06404=1005.162,330.019,338.133,169.528,54.083,160.516
C06405=1005.167,330.267,338.100,169.536,54.078,160.517
C06406=1005.172,330.515,338.067,169.544,54.073,160.517
C06407=1005.178,330.762,338.034,169.552,54.068,160.518
C06408=1005.184,331.010,338.001,169.559,54.064,160.519
C06409=1005.189,331.258,337.969,169.567,54.059,160.519
C06410=1004.884,329.077,337.894,169.480,54.131,160.517
C06411=1004.877,328.829,337.927,169.473,54.136,160.517
C06412=1004.873,328.581,337.959,169.465,54.141,160.516
C06413=1004.867,328.333,337.993,169.457,54.146,160.516
C06414=1004.862,328.086,338.024,169.450,54.151,160.515
C06415=1004.856,327.838,338.058,169.442,54.156,160.515
C06416=1004.851,327.590,338.090,169.435,54.160,160.514
C06417=1004.845,327.342,338.122,169.427,54.165,160.513
C06418=1004.840,327.095,338.155,169.419,54.170,160.513
C06419=1004.835,326.846,338.187,169.412,54.175,160.512
C06420=1004.830,326.599,338.219,169.404,54.180,160.512
C06421=1004.824,326.351,338.252,169.396,54.186,160.511
C06422=1004.820,326.103,338.285,169.389,54.190,160.511
C06423=1004.814,325.855,338.316,169.381,54.195,160.510
C06424=1004.809,325.607,338.350,169.374,54.200,160.510
C06425=1004.803,325.360,338.381,169.366,54.205,160.509
C06426=1004.799,325.112,338.414,169.359,54.210,160.509
C06427=1004.792,324.824,338.452,169.350,54.216,160.508
C06428=1004.787,324.536,338.489,169.341,54.222,160.508
C06429=1004.780,324.247,338.527,169.333,54.228,160.507
C06430=1004.774,323.959,338.563,169.323,54.233,160.506
C06431=1004.769,323.712,338.595,169.316,54.239,160.506
C06432=1004.763,323.463,338.627,169.309,54.244,160.505
C06433=1004.758,323.216,338.659,169.300,54.249,160.505
C06434=1004.753,322.968,338.691,169.293,54.254,160.504
C06435=1004.747,322.719,338.722,169.286,54.259,160.504
C06436=1004.742,322.472,338.754,169.278,54.264,160.503
C06437=1004.737,322.224,338.785,169.271,54.269,160.503
C06438=1004.731,321.977,338.817,169.263,54.274,160.502
C06439=1004.725,321.728,338.848,169.256,54.280,160.502
C06440=1004.721,321.480,338.881,169.248,54.285,160.501
C06441=1004.715,321.233,338.912,169.241,54.289,160.501
C06442=1004.710,320.984,338.943,169.233,54.295,160.501
C06443=1004.705,320.737,338.975,169.226,54.299,160.500
C06444=1004.700,320.489,339.006,169.219,54.305,160.500
C06445=1004.695,320.240,339.038,169.212,54.310,160.499
C06446=1004.690,319.992,339.069,169.204,54.315,160.499
C06447=1004.684,319.745,339.101,169.197,54.320,160.498
C06448=1004.679,319.497,339.133,169.189,54.326,160.498
C06449=1004.674,319.249,339.164,169.182,54.330,160.497
C06450=1004.669,319.001,339.195,169.174,54.336,160.497
C06451=1004.664,318.753,339.227,169.168,54.341,160.497
C06452=1004.659,318.505,339.258,169.160,54.346,160.496
C06453=1004.654,318.257,339.289,169.153,54.352,160.496
C06454=1004.648,318.009,339.320,169.145,54.357,160.495
C06455=1004.643,317.762,339.352,169.138,54.362,160.495
C06456=1004.639,317.513,339.384,169.130,54.367,160.494
C06457=1004.634,317.265,339.415,169.124,54.372,160.494
C06458=1004.628,317.018,339.446,169.116,54.378,160.494
C06459=1004.623,316.770,339.477,169.109,54.383,160.493
C06460=1004.618,316.521,339.508,169.101,54.388,160.493
C06461=1004.614,316.273,339.540,169.095,54.394,160.492
C06462=1004.608,316.025,339.571,169.087,54.398,160.492
C06463=1004.603,315.777,339.602,169.080,54.404,160.491
C06464=1004.599,315.530,339.633,169.073,54.409,160.491
C06465=1004.594,315.282,339.664,169.065,54.414,160.491
C06466=1004.589,315.034,339.696,169.058,54.420,160.490
C06467=1004.584,314.786,339.727,169.052,54.425,160.490
C06468=1004.579,314.538,339.758,169.044,54.431,160.490
C06469=1004.574,314.290,339.789,169.037,54.435,160.489
C06470=1004.569,314.042,339.819,169.029,54.441,160.489
C06471=1004.564,313.794,339.850,169.023,54.446,160.488
C06472=1004.560,313.546,339.882,169.016,54.452,160.488
C06473=1004.555,313.297,339.913,169.008,54.457,160.488
C06474=1004.550,313.050,339.943,169.001,54.462,160.487
C06475=1004.545,312.802,339.974,168.995,54.467,160.487
C06476=1004.540,312.554,340.005,168.987,54.473,160.487
C06477=1004.536,312.306,340.037,168.980,54.478,160.486
C06478=1004.531,312.058,340.067,168.973,54.484,160.486
C06479=1004.526,311.810,340.098,168.966,54.489,160.485
C06480=1004.522,311.562,340.129,168.959,54.494,160.485
C06481=1004.517,311.314,340.160,168.951,54.500,160.485
C06482=1004.512,311.066,340.192,168.945,54.505,160.484
C06483=1004.508,310.818,340.222,168.938,54.510,160.484
C06484=1004.503,310.570,340.252,168.931,54.516,160.484
C06485=1004.499,310.322,340.283,168.924,54.521,160.483
C06486=1004.494,310.074,340.314,168.917,54.527,160.483
C06487=1004.487,309.706,340.360,168.906,54.535,160.482
C06488=1004.480,309.337,340.405,168.896,54.543,160.482
C06489=1004.474,308.969,340.451,168.886,54.551,160.481
C06490=1004.466,308.572,340.500,168.876,54.559,160.481
C06491=1004.220,309.003,340.080,168.869,54.574,160.483
C06492=1004.225,309.281,340.047,168.877,54.568,160.483
C06493=1004.229,309.558,340.012,168.884,54.562,160.484
C06494=1004.235,309.836,339.978,168.893,54.556,160.484
C06495=1004.240,310.113,339.944,168.901,54.550,160.485
C06496=1004.245,310.362,339.912,168.907,54.545,160.485
C06497=1004.249,310.610,339.882,168.915,54.539,160.485
C06498=1004.254,310.858,339.851,168.921,54.534,160.486
C06499=1004.258,311.106,339.821,168.928,54.529,160.486
C06500=1004.263,311.354,339.790,168.935,54.523,160.486
C06501=1004.268,311.602,339.758,168.943,54.518,160.487
C06502=1004.272,311.850,339.728,168.949,54.513,160.487
C06503=1004.277,312.098,339.697,168.956,54.508,160.487
C06504=1004.281,312.346,339.667,168.964,54.502,160.488
C06505=1004.286,312.594,339.636,168.971,54.497,160.488
C06506=1004.291,312.842,339.604,168.977,54.492,160.489
C06507=1004.296,313.090,339.573,168.985,54.486,160.489
C06508=1004.300,313.338,339.543,168.992,54.481,160.489
C06509=1004.305,313.586,339.512,168.999,54.476,160.490
C06510=1004.311,313.834,339.481,169.007,54.471,160.490
C06511=1004.315,314.082,339.450,169.013,54.465,160.491
C06512=1004.319,314.330,339.419,169.020,54.460,160.491
C06513=1004.324,314.578,339.388,169.028,54.455,160.492
C06514=1004.330,314.826,339.356,169.035,54.450,160.492
C06515=1004.335,315.074,339.325,169.042,54.444,160.492
C06516=1004.339,315.321,339.295,169.049,54.439,160.493
C06517=1004.344,315.570,339.263,169.056,54.434,160.493
C06518=1004.349,315.818,339.232,169.064,54.428,160.493
C06519=1004.354,316.066,339.201,169.071,54.424,160.494
C06520=1004.359,316.313,339.170,169.077,54.418,160.494
C06521=1004.364,316.562,339.139,169.085,54.413,160.495
C06522=1004.368,316.809,339.108,169.092,54.408,160.495
C06523=1004.373,317.057,339.077,169.100,54.402,160.496
C06524=1004.379,317.305,339.045,169.107,54.398,160.496
C06525=1004.384,317.553,339.014,169.114,54.392,160.496
C06526=1004.389,317.801,338.983,169.122,54.387,160.497
C06527=1004.393,318.049,338.951,169.128,54.382,160.497
C06528=1004.398,318.297,338.920,169.136,54.377,160.498
C06529=1004.404,318.545,338.889,169.143,54.372,160.498
C06530=1004.409,318.793,338.857,169.151,54.367,160.499
C06531=1004.414,319.041,338.826,169.158,54.361,160.499
C06532=1004.419,319.288,338.795,169.166,54.356,160.500
C06533=1004.424,319.537,338.763,169.172,54.351,160.500
C06534=1004.429,319.785,338.732,169.181,54.346,160.501
C06535=1004.434,320.033,338.700,169.187,54.341,160.501
C06536=1004.439,320.281,338.670,169.195,54.336,160.502
C06537=1004.445,320.529,338.638,169.202,54.331,160.502
C06538=1004.450,320.777,338.605,169.209,54.326,160.502
C06539=1004.455,321.025,338.574,169.217,54.321,160.503
C06540=1004.460,321.272,338.543,169.224,54.315,160.503
C06541=1004.465,321.520,338.512,169.232,54.310,160.504
C06542=1004.471,321.768,338.480,169.240,54.305,160.505
C06543=1004.476,322.017,338.447,169.247,54.300,160.505
C06544=1004.481,322.265,338.416,169.255,54.295,160.505
C06545=1004.487,322.512,338.385,169.262,54.290,160.506
C06546=1004.492,322.760,338.353,169.270,54.285,160.506
C06547=1004.498,323.009,338.322,169.277,54.280,160.507
C06548=1004.503,323.256,338.290,169.285,54.275,160.507
C06549=1004.508,323.504,338.258,169.291,54.270,160.508
C06550=1004.513,323.751,338.226,169.300,54.265,160.508
C06551=1004.519,324.000,338.195,169.307,54.260,160.509
C06552=1004.524,324.237,338.164,169.315,54.255,160.510
C06553=1004.528,324.475,338.134,169.322,54.251,160.510
C06554=1004.534,324.713,338.102,169.328,54.245,160.510
C06555=1004.538,324.950,338.072,169.336,54.241,160.511
C06556=1004.544,325.188,338.041,169.343,54.236,160.511
C06557=1004.548,325.425,338.010,169.350,54.231,160.512
C06558=1004.554,325.663,337.979,169.358,54.226,160.512
C06559=1004.558,325.901,337.948,169.365,54.222,160.513
C06560=1004.564,326.149,337.915,169.372,54.217,160.513
C06561=1004.569,326.396,337.883,169.380,54.212,160.514
C06562=1004.574,326.644,337.851,169.388,54.207,160.515
C06563=1004.580,326.892,337.819,169.396,54.203,160.515
C06564=1004.277,324.708,337.740,169.311,54.272,160.513
C06565=1004.270,324.374,337.783,169.301,54.278,160.512
C06566=1004.263,324.040,337.826,169.291,54.285,160.511
C06567=1004.258,323.792,337.857,169.283,54.290,160.511
C06568=1004.253,323.544,337.890,169.276,54.295,160.510
C06569=1004.248,323.296,337.921,169.268,54.300,160.510
C06570=1004.242,323.048,337.953,169.261,54.305,160.509
C06571=1004.237,322.800,337.984,169.253,54.310,160.509
C06572=1004.231,322.553,338.016,169.246,54.315,160.508
C06573=1004.226,322.305,338.048,169.238,54.320,160.508
C06574=1004.221,322.057,338.079,169.231,54.325,160.507
C06575=1004.215,321.808,338.111,169.223,54.330,160.506
C06576=1004.210,321.560,338.142,169.216,54.335,160.506
C06577=1004.205,321.313,338.174,169.208,54.340,160.506
C06578=1004.200,321.065,338.205,169.201,54.345,160.505
C06579=1004.195,320.817,338.237,169.193,54.351,160.505
C06580=1004.190,320.569,338.269,169.186,54.355,160.504
C06581=1004.185,320.321,338.300,169.178,54.360,160.503
C06582=1004.179,320.074,338.331,169.171,54.366,160.503
C06583=1004.174,319.825,338.362,169.163,54.371,160.503
C06584=1004.170,319.577,338.394,169.157,54.376,160.502
C06585=1004.165,319.330,338.425,169.150,54.380,160.502
C06586=1004.159,319.081,338.456,169.141,54.386,160.501
C06587=1004.154,318.834,338.488,169.135,54.391,160.501
C06588=1004.149,318.586,338.519,169.127,54.396,160.500
C06589=1004.145,318.337,338.550,169.120,54.401,160.500
C06590=1004.139,318.090,338.582,169.112,54.406,160.499
C06591=1004.134,317.842,338.613,169.105,54.411,160.499
C06592=1004.129,317.594,338.644,169.098,54.416,160.498
C06593=1004.124,317.346,338.676,169.091,54.422,160.498
C06594=1004.119,317.098,338.707,169.083,54.426,160.498
C06595=1004.114,316.849,338.738,169.076,54.432,160.497
C06596=1004.109,316.601,338.769,169.069,54.437,160.497
C06597=1004.104,316.353,338.800,169.062,54.442,160.496
C06598=1004.099,316.106,338.831,169.054,54.447,160.496
C06599=1004.094,315.858,338.862,169.047,54.452,160.495
C06600=1004.090,315.610,338.894,169.040,54.457,160.495
C06601=1004.085,315.362,338.925,169.033,54.463,160.494
C06602=1004.080,315.114,338.956,169.025,54.467,160.494
C06603=1004.075,314.865,338.987,169.019,54.473,160.494
C06604=1004.070,314.618,339.017,169.011,54.478,160.493
C06605=1004.066,314.370,339.049,169.004,54.483,160.493
C06606=1004.061,314.121,339.080,168.997,54.488,160.492
C06607=1004.056,313.874,339.110,168.990,54.494,160.492
C06608=1004.051,313.626,339.141,168.983,54.499,160.491
C06609=1004.046,313.378,339.172,168.976,54.504,160.491
C06610=1004.042,313.130,339.203,168.968,54.510,160.491
C06611=1004.037,312.882,339.234,168.961,54.514,160.490
C06612=1004.032,312.634,339.265,168.955,54.520,160.490
C06613=1004.028,312.386,339.296,168.947,54.526,160.490
C06614=1004.023,312.138,339.327,168.940,54.530,160.489
C06615=1004.018,311.890,339.358,168.933,54.535,160.489
C06616=1004.014,311.642,339.388,168.926,54.541,160.488
C06617=1004.009,311.393,339.419,168.919,54.547,160.488
C06618=1004.005,311.146,339.450,168.912,54.551,160.487
C06619=1004.001,310.934,339.476,168.906,54.556,160.487
C06620=1003.996,310.722,339.502,168.900,54.560,160.487
C06621=1003.993,310.510,339.529,168.894,54.565,160.486
C06622=1003.989,310.298,339.555,168.888,54.569,160.486
C06623=1003.985,310.087,339.581,168.882,54.574,160.486
C06624=1003.981,309.874,339.607,168.877,54.579,160.486
C06625=1003.977,309.663,339.633,168.871,54.583,160.485
C06626=1003.974,309.451,339.659,168.864,54.587,160.485
C06627=1003.727,309.889,339.240,168.858,54.600,160.487
C06628=1003.731,310.101,339.214,168.866,54.596,160.487
C06629=1003.735,310.315,339.188,168.872,54.591,160.487
C06630=1003.739,310.528,339.161,168.877,54.586,160.488
C06631=1003.743,310.741,339.134,168.883,54.582,160.488
C06632=1003.747,310.954,339.109,168.890,54.578,160.488
C06633=1003.750,311.167,339.081,168.895,54.573,160.489
C06634=1003.754,311.381,339.055,168.901,54.569,160.489
C06635=1003.758,311.594,339.029,168.907,54.565,160.489
C06636=1003.763,311.842,338.998,168.914,54.559,160.490
C06637=1003.768,312.090,338.967,168.922,54.553,160.490
C06638=1003.773,312.338,338.936,168.929,54.549,160.491
C06639=1003.777,312.587,338.906,168.935,54.543,160.491
C06640=1003.782,312.835,338.875,168.942,54.539,160.492
C06641=1003.786,313.082,338.844,168.950,54.533,160.492
C06642=1003.791,313.330,338.813,168.957,54.528,160.492
C06643=1003.796,313.578,338.782,168.964,54.523,160.493
C06644=1003.800,313.826,338.751,168.972,54.517,160.493
C06645=1003.805,314.074,338.720,168.979,54.513,160.494
C06646=1003.810,314.322,338.689,168.985,54.507,160.494
C06647=1003.815,314.570,338.659,168.992,54.502,160.494
C06648=1003.820,314.818,338.628,169.000,54.497,160.495
C06649=1003.824,315.066,338.596,169.007,54.492,160.495
C06650=1003.829,315.314,338.565,169.014,54.487,160.496
C06651=1003.834,315.562,338.535,169.021,54.481,160.496
C06652=1003.839,315.810,338.504,169.029,54.477,160.497
C06653=1003.844,316.058,338.473,169.035,54.472,160.497
C06654=1003.848,316.307,338.441,169.043,54.466,160.498
C06655=1003.853,316.555,338.410,169.050,54.461,160.498
C06656=1003.858,316.802,338.379,169.057,54.457,160.499
C06657=1003.863,317.050,338.348,169.065,54.451,160.499
C06658=1003.868,317.298,338.317,169.072,54.446,160.499
C06659=1003.872,317.546,338.286,169.080,54.441,160.500
C06660=1003.878,317.794,338.255,169.087,54.436,160.500
C06661=1003.883,318.042,338.223,169.094,54.431,160.501
C06662=1003.888,318.290,338.192,169.101,54.425,160.501
C06663=1003.893,318.538,338.161,169.108,54.421,160.502
C06664=1003.898,318.786,338.129,169.116,54.416,160.502
C06665=1003.903,319.034,338.098,169.123,54.411,160.503
C06666=1003.908,319.282,338.067,169.130,54.406,160.503
C06667=1003.913,319.530,338.035,169.138,54.401,160.504
C06668=1003.918,319.778,338.004,169.145,54.396,160.504
C06669=1003.923,320.026,337.973,169.153,54.391,160.505
C06670=1003.928,320.274,337.941,169.160,54.386,160.505
C06671=1003.933,320.522,337.910,169.167,54.381,160.506
C06672=1003.939,320.770,337.879,169.175,54.376,160.506
C06673=1003.944,321.018,337.848,169.182,54.371,160.507
C06674=1003.949,321.265,337.816,169.190,54.365,160.507
C06675=1003.953,321.514,337.784,169.197,54.361,160.508
C06676=1003.959,321.761,337.753,169.205,54.356,160.508
C06677=1003.964,322.009,337.722,169.212,54.351,160.509
C06678=1003.969,322.257,337.690,169.220,54.345,160.509
C06679=1003.975,322.505,337.658,169.227,54.341,160.510
C06680=1003.673,320.298,337.574,169.144,54.408,160.507
C06681=1003.668,320.050,337.605,169.136,54.413,160.506
C06682=1003.663,319.802,337.637,169.129,54.419,160.506
C06683=1003.658,319.554,337.668,169.122,54.423,160.506
C06684=1003.653,319.306,337.700,169.114,54.428,160.505
C06685=1003.648,319.058,337.731,169.107,54.433,160.504
C06686=1003.643,318.810,337.762,169.099,54.439,160.504
C06687=1003.638,318.562,337.793,169.092,54.443,160.503
C06688=1003.633,318.314,337.825,169.085,54.448,160.503
C06689=1003.628,318.066,337.856,169.077,54.454,160.502
C06690=1003.624,317.818,337.887,169.070,54.458,160.502
C06691=1003.619,317.570,337.918,169.063,54.463,160.501
C06692=1003.613,317.323,337.949,169.056,54.469,160.501
C06693=1003.608,317.075,337.980,169.048,54.473,160.500
C06694=1003.603,316.827,338.011,169.041,54.478,160.500
C06695=1003.599,316.578,338.043,169.034,54.484,160.500
C06696=1003.594,316.331,338.073,169.027,54.488,160.499
C06697=1003.589,316.083,338.104,169.020,54.494,160.499
C06698=1003.584,315.834,338.135,169.012,54.499,160.498
C06699=1003.579,315.586,338.166,169.005,54.504,160.498
C06700=1003.575,315.339,338.197,168.998,54.509,160.497
C06701=1003.570,315.090,338.228,168.990,54.514,160.497
C06702=1003.565,314.842,338.259,168.983,54.519,160.496
C06703=1003.560,314.594,338.290,168.976,54.524,160.496
C06704=1003.556,314.347,338.321,168.970,54.529,160.495
C06705=1003.551,314.098,338.352,168.961,54.534,160.495
C06706=1003.546,313.850,338.383,168.955,54.539,160.494
C06707=1003.542,313.603,338.414,168.948,54.544,160.494
C06708=1003.537,313.355,338.445,168.941,54.549,160.494
C06709=1003.532,313.107,338.475,168.933,54.555,160.493
C06710=1003.528,312.859,338.507,168.926,54.560,160.493
C06711=1003.523,312.610,338.537,168.920,54.565,160.492
C06712=1003.519,312.363,338.568,168.912,54.570,160.492
C06713=1003.514,312.114,338.599,168.905,54.575,160.491
C06714=1003.509,311.867,338.629,168.898,54.580,160.491
C06715=1003.505,311.619,338.661,168.891,54.585,160.491
C06716=1003.501,311.370,338.691,168.884,54.591,160.490
C06717=1003.495,311.106,338.723,168.876,54.596,160.490
C06718=1003.491,310.842,338.756,168.869,54.601,160.489
C06719=1003.486,310.577,338.789,168.861,54.607,160.489
C06720=1003.481,310.313,338.821,168.854,54.612,160.488
C06721=1003.234,310.726,338.404,168.849,54.624,160.490
C06722=1003.241,311.080,338.362,168.859,54.617,160.490
C06723=1003.247,311.432,338.318,168.869,54.610,160.491
C06724=1003.254,311.786,338.273,168.879,54.603,160.492
C06725=1003.260,312.139,338.230,168.889,54.595,160.492
C06726=1003.265,312.387,338.200,168.896,54.590,160.493
C06727=1003.269,312.635,338.168,168.903,54.585,160.493
C06728=1003.274,312.882,338.138,168.910,54.580,160.494
C06729=1003.278,313.131,338.108,168.918,54.575,160.494
C06730=1003.284,313.379,338.077,168.925,54.570,160.495
C06731=1003.288,313.627,338.046,168.931,54.565,160.495
C06732=1003.292,313.875,338.014,168.939,54.560,160.496
C06733=1003.297,314.123,337.984,168.945,54.555,160.496
C06734=1003.302,314.371,337.953,168.953,54.550,160.497
C06735=1003.307,314.619,337.922,168.960,54.545,160.497
C06736=1003.311,314.866,337.891,168.967,54.540,160.497
C06737=1003.316,315.115,337.860,168.974,54.535,160.498
C06738=1003.321,315.363,337.829,168.982,54.529,160.498
C06739=1003.325,315.610,337.798,168.989,54.525,160.499
C06740=1003.330,315.858,337.767,168.996,54.520,160.499
C06741=1003.336,316.107,337.736,169.004,54.514,160.500
C06742=1003.340,316.355,337.705,169.011,54.510,160.500
C06743=1003.344,316.602,337.674,169.017,54.504,160.501
C06744=1003.349,316.851,337.643,169.025,54.500,160.501
C06745=1003.355,317.099,337.612,169.033,54.495,160.502
C06746=1003.360,317.347,337.582,169.039,54.489,160.502
C06747=1003.364,317.595,337.550,169.046,54.485,160.503
C06748=1003.368,317.843,337.519,169.055,54.480,160.503
C06749=1003.374,318.091,337.488,169.062,54.475,160.504
C06750=1003.076,315.884,337.399,168.980,54.540,160.500
C06751=1003.072,315.636,337.431,168.973,54.544,160.500
C06752=1003.067,315.388,337.462,168.966,54.550,160.499
C06753=1003.062,315.140,337.492,168.958,54.555,160.499
C06754=1003.057,314.892,337.523,168.951,54.559,160.498
C06755=1003.053,314.643,337.554,168.945,54.565,160.498
C06756=1003.049,314.396,337.585,168.937,54.570,160.497
C06757=1003.044,314.147,337.616,168.929,54.574,160.497
C06758=1003.039,313.900,337.646,168.923,54.580,160.497
C06759=1003.034,313.652,337.677,168.916,54.584,160.496
C06760=1003.029,313.404,337.708,168.909,54.590,160.496
C06761=1003.026,313.155,337.739,168.901,54.595,160.495
C06762=1003.021,312.907,337.770,168.894,54.600,160.495
C06763=1003.016,312.685,337.797,168.888,54.604,160.494
C06764=1003.013,312.463,337.824,168.882,54.608,160.494
C06765=1003.008,312.241,337.852,168.875,54.613,160.493
C06766=1003.004,312.018,337.880,168.869,54.617,160.493
C06767=1003.000,311.797,337.907,168.863,54.622,160.493
C06768=1002.996,311.574,337.934,168.856,54.627,160.492
C06769=1002.992,311.351,337.961,168.850,54.631,160.492
C06770=1002.988,311.130,337.989,168.844,54.635,160.491
C06771=1002.742,311.523,337.575,168.838,54.647,160.493
C06772=1002.747,311.813,337.539,168.846,54.641,160.493
C06773=1002.752,312.104,337.503,168.855,54.636,160.494
C06774=1002.758,312.394,337.468,168.863,54.629,160.494
C06775=1002.762,312.685,337.431,168.872,54.623,160.495
C06776=1002.767,312.933,337.400,168.879,54.619,160.495
C06777=1002.771,313.181,337.370,168.886,54.613,160.496
C06778=1002.777,313.429,337.340,168.893,54.609,160.496
C06779=1002.781,313.677,337.309,168.899,54.603,160.497
C06780=952.366,450.117,285.118,168.899,54.603,160.497
///USER 0
///POSTYPE ROBOT
///RECTAN
C06781=725.000,0.000,388.500,-180.000,-0.000,0.000
//INST
///DATE 2021/06/25 14:50
///ATTR SC,RW,RJ
////FRAME ROBOT
///GROUP1 RB1
NOP
MOVL C00000 V=800.0 PL=0
MOVL C00001 V=800.0 PL=0
MOVL C00002 V=800.0 PL=0
MOVL C00003 V=800.0 PL=0
MOVL C00004 V=800.0 PL=0
MOVL C00005 V=800.0 PL=0
MOVL C00006 V=800.0 PL=0
MOVL C00007 V=800.0 PL=0
MOVL C00008 V=800.0 PL=0
MOVL C00009 V=800.0 PL=0
MOVL C00010 V=800.0 PL=0
MOVL C00011 V=800.0 PL=0
MOVL C00012 V=800.0 PL=0
MOVL C00013 V=800.0 PL=0
MOVL C00014 V=800.0 PL=0
MOVL C00015 V=800.0 PL=0
MOVL C00016 V=800.0 PL=0
MOVL C00017 V=800.0 PL=0
MOVL C00018 V=800.0 PL=0
MOVL C00019 V=800.0 PL=0
MOVL C00020 V=800.0 PL=0
MOVL C00021 V=800.0 PL=0
MOVL C00022 V=800.0 PL=0
MOVL C00023 V=800.0 PL=0
MOVL C00024 V=800.0 PL=0
MOVL C00025 V=800.0 PL=0
MOVL C00026 V=800.0 PL=0
MOVL C00027 V=800.0 PL=0
MOVL C00028 V=800.0 PL=0
MOVL C00029 V=800.0 PL=0
MOVL C00030 V=800.0 PL=0
MOVL C00031 V=800.0 PL=0
MOVL C00032 V=800.0 PL=0
MOVL C00033 V=800.0 PL=0
MOVL C00034 V=800.0 PL=0
MOVL C00035 V=800.0 PL=0
MOVL C00036 V=800.0 PL=0
MOVL C00037 V=800.0 PL=0
MOVL C00038 V=800.0 PL=0
MOVL C00039 V=800.0 PL=0
MOVL C00040 V=800.0 PL=0
MOVL C00041 V=800.0 PL=0
MOVL C00042 V=800.0 PL=0
MOVL C00043 V=800.0 PL=0
MOVL C00044 V=800.0 PL=0
MOVL C00045 V=800.0 PL=0
MOVL C00046 V=800.0 PL=0
MOVL C00047 V=800.0 PL=0
MOVL C00048 V=800.0 PL=0
MOVL C00049 V=800.0 PL=0
MOVL C00050 V=800.0 PL=0
MOVL C00051 V=800.0 PL=0
MOVL C00052 V=800.0 PL=0
MOVL C00053 V=800.0 PL=0
MOVL C00054 V=800.0 PL=0
MOVL C00055 V=800.0 PL=0
MOVL C00056 V=800.0 PL=0
MOVL C00057 V=800.0 PL=0
MOVL C00058 V=800.0 PL=0
MOVL C00059 V=800.0 PL=0
MOVL C00060 V=800.0 PL=0
MOVL C00061 V=800.0 PL=0
MOVL C00062 V=800.0 PL=0
MOVL C00063 V=800.0 PL=0
MOVL C00064 V=800.0 PL=0
MOVL C00065 V=800.0 PL=0
MOVL C00066 V=800.0 PL=0
MOVL C00067 V=800.0 PL=0
MOVL C00068 V=800.0 PL=0
MOVL C00069 V=800.0 PL=0
MOVL C00070 V=800.0 PL=0
MOVL C00071 V=800.0 PL=0
MOVL C00072 V=800.0 PL=0
MOVL C00073 V=800.0 PL=0
MOVL C00074 V=800.0 PL=0
MOVL C00075 V=800.0 PL=0
MOVL C00076 V=800.0 PL=0
MOVL C00077 V=800.0 PL=0
MOVL C00078 V=800.0 PL=0
MOVL C00079 V=800.0 PL=0
MOVL C00080 V=800.0 PL=0
MOVL C00081 V=800.0 PL=0
MOVL C00082 V=800.0 PL=0
MOVL C00083 V=800.0 PL=0
MOVL C00084 V=800.0 PL=0
MOVL C00085 V=800.0 PL=0
MOVL C00086 V=800.0 PL=0
MOVL C00087 V=800.0 PL=0
MOVL C00088 V=800.0 PL=0
MOVL C00089 V=800.0 PL=0
MOVL C00090 V=800.0 PL=0
MOVL C00091 V=800.0 PL=0
MOVL C00092 V=800.0 PL=0
MOVL C00093 V=800.0 PL=0
MOVL C00094 V=800.0 PL=0
MOVL C00095 V=800.0 PL=0
MOVL C00096 V=800.0 PL=0
MOVL C00097 V=800.0 PL=0
MOVL C00098 V=800.0 PL=0
MOVL C00099 V=800.0 PL=0
MOVL C00100 V=800.0 PL=0
MOVL C00101 V=800.0 PL=0
MOVL C00102 V=800.0 PL=0
MOVL C00103 V=800.0 PL=0
MOVL C00104 V=800.0 PL=0
MOVL C00105 V=800.0 PL=0
MOVL C00106 V=800.0 PL=0
MOVL C00107 V=800.0 PL=0
MOVL C00108 V=800.0 PL=0
MOVL C00109 V=800.0 PL=0
MOVL C00110 V=800.0 PL=0
MOVL C00111 V=800.0 PL=0
MOVL C00112 V=800.0 PL=0
MOVL C00113 V=800.0 PL=0
MOVL C00114 V=800.0 PL=0
MOVL C00115 V=800.0 PL=0
MOVL C00116 V=800.0 PL=0
MOVL C00117 V=800.0 PL=0
MOVL C00118 V=800.0 PL=0
MOVL C00119 V=800.0 PL=0
MOVL C00120 V=800.0 PL=0
MOVL C00121 V=800.0 PL=0
MOVL C00122 V=800.0 PL=0
MOVL C00123 V=800.0 PL=0
MOVL C00124 V=800.0 PL=0
MOVL C00125 V=800.0 PL=0
MOVL C00126 V=800.0 PL=0
MOVL C00127 V=800.0 PL=0
MOVL C00128 V=800.0 PL=0
MOVL C00129 V=800.0 PL=0
MOVL C00130 V=800.0 PL=0
MOVL C00131 V=800.0 PL=0
MOVL C00132 V=800.0 PL=0
MOVL C00133 V=800.0 PL=0
MOVL C00134 V=800.0 PL=0
MOVL C00135 V=800.0 PL=0
MOVL C00136 V=800.0 PL=0
MOVL C00137 V=800.0 PL=0
MOVL C00138 V=800.0 PL=0
MOVL C00139 V=800.0 PL=0
MOVL C00140 V=800.0 PL=0
MOVL C00141 V=800.0 PL=0
MOVL C00142 V=800.0 PL=0
MOVL C00143 V=800.0 PL=0
MOVL C00144 V=800.0 PL=0
MOVL C00145 V=800.0 PL=0
MOVL C00146 V=800.0 PL=0
MOVL C00147 V=800.0 PL=0
MOVL C00148 V=800.0 PL=0
MOVL C00149 V=800.0 PL=0
MOVL C00150 V=800.0 PL=0
MOVL C00151 V=800.0 PL=0
MOVL C00152 V=800.0 PL=0
MOVL C00153 V=800.0 PL=0
MOVL C00154 V=800.0 PL=0
MOVL C00155 V=800.0 PL=0
MOVL C00156 V=800.0 PL=0
MOVL C00157 V=800.0 PL=0
MOVL C00158 V=800.0 PL=0
MOVL C00159 V=800.0 PL=0
MOVL C00160 V=800.0 PL=0
MOVL C00161 V=800.0 PL=0
MOVL C00162 V=800.0 PL=0
MOVL C00163 V=800.0 PL=0
MOVL C00164 V=800.0 PL=0
MOVL C00165 V=800.0 PL=0
MOVL C00166 V=800.0 PL=0
MOVL C00167 V=800.0 PL=0
MOVL C00168 V=800.0 PL=0
MOVL C00169 V=800.0 PL=0
MOVL C00170 V=800.0 PL=0
MOVL C00171 V=800.0 PL=0
MOVL C00172 V=800.0 PL=0
MOVL C00173 V=800.0 PL=0
MOVL C00174 V=800.0 PL=0
MOVL C00175 V=800.0 PL=0
MOVL C00176 V=800.0 PL=0
MOVL C00177 V=800.0 PL=0
MOVL C00178 V=800.0 PL=0
MOVL C00179 V=800.0 PL=0
MOVL C00180 V=800.0 PL=0
MOVL C00181 V=800.0 PL=0
MOVL C00182 V=800.0 PL=0
MOVL C00183 V=800.0 PL=0
MOVL C00184 V=800.0 PL=0
MOVL C00185 V=800.0 PL=0
MOVL C00186 V=800.0 PL=0
MOVL C00187 V=800.0 PL=0
MOVL C00188 V=800.0 PL=0
MOVL C00189 V=800.0 PL=0
MOVL C00190 V=800.0 PL=0
MOVL C00191 V=800.0 PL=0
MOVL C00192 V=800.0 PL=0
MOVL C00193 V=800.0 PL=0
MOVL C00194 V=800.0 PL=0
MOVL C00195 V=800.0 PL=0
MOVL C00196 V=800.0 PL=0
MOVL C00197 V=800.0 PL=0
MOVL C00198 V=800.0 PL=0
MOVL C00199 V=800.0 PL=0
MOVL C00200 V=800.0 PL=0
MOVL C00201 V=800.0 PL=0
MOVL C00202 V=800.0 PL=0
MOVL C00203 V=800.0 PL=0
MOVL C00204 V=800.0 PL=0
MOVL C00205 V=800.0 PL=0
MOVL C00206 V=800.0 PL=0
MOVL C00207 V=800.0 PL=0
MOVL C00208 V=800.0 PL=0
MOVL C00209 V=800.0 PL=0
MOVL C00210 V=800.0 PL=0
MOVL C00211 V=800.0 PL=0
MOVL C00212 V=800.0 PL=0
MOVL C00213 V=800.0 PL=0
MOVL C00214 V=800.0 PL=0
MOVL C00215 V=800.0 PL=0
MOVL C00216 V=800.0 PL=0
MOVL C00217 V=800.0 PL=0
MOVL C00218 V=800.0 PL=0
MOVL C00219 V=800.0 PL=0
MOVL C00220 V=800.0 PL=0
MOVL C00221 V=800.0 PL=0
MOVL C00222 V=800.0 PL=0
MOVL C00223 V=800.0 PL=0
MOVL C00224 V=800.0 PL=0
MOVL C00225 V=800.0 PL=0
MOVL C00226 V=800.0 PL=0
MOVL C00227 V=800.0 PL=0
MOVL C00228 V=800.0 PL=0
MOVL C00229 V=800.0 PL=0
MOVL C00230 V=800.0 PL=0
MOVL C00231 V=800.0 PL=0
MOVL C00232 V=800.0 PL=0
MOVL C00233 V=800.0 PL=0
MOVL C00234 V=800.0 PL=0
MOVL C00235 V=800.0 PL=0
MOVL C00236 V=800.0 PL=0
MOVL C00237 V=800.0 PL=0
MOVL C00238 V=800.0 PL=0
MOVL C00239 V=800.0 PL=0
MOVL C00240 V=800.0 PL=0
MOVL C00241 V=800.0 PL=0
MOVL C00242 V=800.0 PL=0
MOVL C00243 V=800.0 PL=0
MOVL C00244 V=800.0 PL=0
MOVL C00245 V=800.0 PL=0
MOVL C00246 V=800.0 PL=0
MOVL C00247 V=800.0 PL=0
MOVL C00248 V=800.0 PL=0
MOVL C00249 V=800.0 PL=0
MOVL C00250 V=800.0 PL=0
MOVL C00251 V=800.0 PL=0
MOVL C00252 V=800.0 PL=0
MOVL C00253 V=800.0 PL=0
MOVL C00254 V=800.0 PL=0
MOVL C00255 V=800.0 PL=0
MOVL C00256 V=800.0 PL=0
MOVL C00257 V=800.0 PL=0
MOVL C00258 V=800.0 PL=0
MOVL C00259 V=800.0 PL=0
MOVL C00260 V=800.0 PL=0
MOVL C00261 V=800.0 PL=0
MOVL C00262 V=800.0 PL=0
MOVL C00263 V=800.0 PL=0
MOVL C00264 V=800.0 PL=0
MOVL C00265 V=800.0 PL=0
MOVL C00266 V=800.0 PL=0
MOVL C00267 V=800.0 PL=0
MOVL C00268 V=800.0 PL=0
MOVL C00269 V=800.0 PL=0
MOVL C00270 V=800.0 PL=0
MOVL C00271 V=800.0 PL=0
MOVL C00272 V=800.0 PL=0
MOVL C00273 V=800.0 PL=0
MOVL C00274 V=800.0 PL=0
MOVL C00275 V=800.0 PL=0
MOVL C00276 V=800.0 PL=0
MOVL C00277 V=800.0 PL=0
MOVL C00278 V=800.0 PL=0
MOVL C00279 V=800.0 PL=0
MOVL C00280 V=800.0 PL=0
MOVL C00281 V=800.0 PL=0
MOVL C00282 V=800.0 PL=0
MOVL C00283 V=800.0 PL=0
MOVL C00284 V=800.0 PL=0
MOVL C00285 V=800.0 PL=0
MOVL C00286 V=800.0 PL=0
MOVL C00287 V=800.0 PL=0
MOVL C00288 V=800.0 PL=0
MOVL C00289 V=800.0 PL=0
MOVL C00290 V=800.0 PL=0
MOVL C00291 V=800.0 PL=0
MOVL C00292 V=800.0 PL=0
MOVL C00293 V=800.0 PL=0
MOVL C00294 V=800.0 PL=0
MOVL C00295 V=800.0 PL=0
MOVL C00296 V=800.0 PL=0
MOVL C00297 V=800.0 PL=0
MOVL C00298 V=800.0 PL=0
MOVL C00299 V=800.0 PL=0
MOVL C00300 V=800.0 PL=0
MOVL C00301 V=800.0 PL=0
MOVL C00302 V=800.0 PL=0
MOVL C00303 V=800.0 PL=0
MOVL C00304 V=800.0 PL=0
MOVL C00305 V=800.0 PL=0
MOVL C00306 V=800.0 PL=0
MOVL C00307 V=800.0 PL=0
MOVL C00308 V=800.0 PL=0
MOVL C00309 V=800.0 PL=0
MOVL C00310 V=800.0 PL=0
MOVL C00311 V=800.0 PL=0
MOVL C00312 V=800.0 PL=0
MOVL C00313 V=800.0 PL=0
MOVL C00314 V=800.0 PL=0
MOVL C00315 V=800.0 PL=0
MOVL C00316 V=800.0 PL=0
MOVL C00317 V=800.0 PL=0
MOVL C00318 V=800.0 PL=0
MOVL C00319 V=800.0 PL=0
MOVL C00320 V=800.0 PL=0
MOVL C00321 V=800.0 PL=0
MOVL C00322 V=800.0 PL=0
MOVL C00323 V=800.0 PL=0
MOVL C00324 V=800.0 PL=0
MOVL C00325 V=800.0 PL=0
MOVL C00326 V=800.0 PL=0
MOVL C00327 V=800.0 PL=0
MOVL C00328 V=800.0 PL=0
MOVL C00329 V=800.0 PL=0
MOVL C00330 V=800.0 PL=0
MOVL C00331 V=800.0 PL=0
MOVL C00332 V=800.0 PL=0
MOVL C00333 V=800.0 PL=0
MOVL C00334 V=800.0 PL=0
MOVL C00335 V=800.0 PL=0
MOVL C00336 V=800.0 PL=0
MOVL C00337 V=800.0 PL=0
MOVL C00338 V=800.0 PL=0
MOVL C00339 V=800.0 PL=0
MOVL C00340 V=800.0 PL=0
MOVL C00341 V=800.0 PL=0
MOVL C00342 V=800.0 PL=0
MOVL C00343 V=800.0 PL=0
MOVL C00344 V=800.0 PL=0
MOVL C00345 V=800.0 PL=0
MOVL C00346 V=800.0 PL=0
MOVL C00347 V=800.0 PL=0
MOVL C00348 V=800.0 PL=0
MOVL C00349 V=800.0 PL=0
MOVL C00350 V=800.0 PL=0
MOVL C00351 V=800.0 PL=0
MOVL C00352 V=800.0 PL=0
MOVL C00353 V=800.0 PL=0
MOVL C00354 V=800.0 PL=0
MOVL C00355 V=800.0 PL=0
MOVL C00356 V=800.0 PL=0
MOVL C00357 V=800.0 PL=0
MOVL C00358 V=800.0 PL=0
MOVL C00359 V=800.0 PL=0
MOVL C00360 V=800.0 PL=0
MOVL C00361 V=800.0 PL=0
MOVL C00362 V=800.0 PL=0
MOVL C00363 V=800.0 PL=0
MOVL C00364 V=800.0 PL=0
MOVL C00365 V=800.0 PL=0
MOVL C00366 V=800.0 PL=0
MOVL C00367 V=800.0 PL=0
MOVL C00368 V=800.0 PL=0
MOVL C00369 V=800.0 PL=0
MOVL C00370 V=800.0 PL=0
MOVL C00371 V=800.0 PL=0
MOVL C00372 V=800.0 PL=0
MOVL C00373 V=800.0 PL=0
MOVL C00374 V=800.0 PL=0
MOVL C00375 V=800.0 PL=0
MOVL C00376 V=800.0 PL=0
MOVL C00377 V=800.0 PL=0
MOVL C00378 V=800.0 PL=0
MOVL C00379 V=800.0 PL=0
MOVL C00380 V=800.0 PL=0
MOVL C00381 V=800.0 PL=0
MOVL C00382 V=800.0 PL=0
MOVL C00383 V=800.0 PL=0
MOVL C00384 V=800.0 PL=0
MOVL C00385 V=800.0 PL=0
MOVL C00386 V=800.0 PL=0
MOVL C00387 V=800.0 PL=0
MOVL C00388 V=800.0 PL=0
MOVL C00389 V=800.0 PL=0
MOVL C00390 V=800.0 PL=0
MOVL C00391 V=800.0 PL=0
MOVL C00392 V=800.0 PL=0
MOVL C00393 V=800.0 PL=0
MOVL C00394 V=800.0 PL=0
MOVL C00395 V=800.0 PL=0
MOVL C00396 V=800.0 PL=0
MOVL C00397 V=800.0 PL=0
MOVL C00398 V=800.0 PL=0
MOVL C00399 V=800.0 PL=0
MOVL C00400 V=800.0 PL=0
MOVL C00401 V=800.0 PL=0
MOVL C00402 V=800.0 PL=0
MOVL C00403 V=800.0 PL=0
MOVL C00404 V=800.0 PL=0
MOVL C00405 V=800.0 PL=0
MOVL C00406 V=800.0 PL=0
MOVL C00407 V=800.0 PL=0
MOVL C00408 V=800.0 PL=0
MOVL C00409 V=800.0 PL=0
MOVL C00410 V=800.0 PL=0
MOVL C00411 V=800.0 PL=0
MOVL C00412 V=800.0 PL=0
MOVL C00413 V=800.0 PL=0
MOVL C00414 V=800.0 PL=0
MOVL C00415 V=800.0 PL=0
MOVL C00416 V=800.0 PL=0
MOVL C00417 V=800.0 PL=0
MOVL C00418 V=800.0 PL=0
MOVL C00419 V=800.0 PL=0
MOVL C00420 V=800.0 PL=0
MOVL C00421 V=800.0 PL=0
MOVL C00422 V=800.0 PL=0
MOVL C00423 V=800.0 PL=0
MOVL C00424 V=800.0 PL=0
MOVL C00425 V=800.0 PL=0
MOVL C00426 V=800.0 PL=0
MOVL C00427 V=800.0 PL=0
MOVL C00428 V=800.0 PL=0
MOVL C00429 V=800.0 PL=0
MOVL C00430 V=800.0 PL=0
MOVL C00431 V=800.0 PL=0
MOVL C00432 V=800.0 PL=0
MOVL C00433 V=800.0 PL=0
MOVL C00434 V=800.0 PL=0
MOVL C00435 V=800.0 PL=0
MOVL C00436 V=800.0 PL=0
MOVL C00437 V=800.0 PL=0
MOVL C00438 V=800.0 PL=0
MOVL C00439 V=800.0 PL=0
MOVL C00440 V=800.0 PL=0
MOVL C00441 V=800.0 PL=0
MOVL C00442 V=800.0 PL=0
MOVL C00443 V=800.0 PL=0
MOVL C00444 V=800.0 PL=0
MOVL C00445 V=800.0 PL=0
MOVL C00446 V=800.0 PL=0
MOVL C00447 V=800.0 PL=0
MOVL C00448 V=800.0 PL=0
MOVL C00449 V=800.0 PL=0
MOVL C00450 V=800.0 PL=0
MOVL C00451 V=800.0 PL=0
MOVL C00452 V=800.0 PL=0
MOVL C00453 V=800.0 PL=0
MOVL C00454 V=800.0 PL=0
MOVL C00455 V=800.0 PL=0
MOVL C00456 V=800.0 PL=0
MOVL C00457 V=800.0 PL=0
MOVL C00458 V=800.0 PL=0
MOVL C00459 V=800.0 PL=0
MOVL C00460 V=800.0 PL=0
MOVL C00461 V=800.0 PL=0
MOVL C00462 V=800.0 PL=0
MOVL C00463 V=800.0 PL=0
MOVL C00464 V=800.0 PL=0
MOVL C00465 V=800.0 PL=0
MOVL C00466 V=800.0 PL=0
MOVL C00467 V=800.0 PL=0
MOVL C00468 V=800.0 PL=0
MOVL C00469 V=800.0 PL=0
MOVL C00470 V=800.0 PL=0
MOVL C00471 V=800.0 PL=0
MOVL C00472 V=800.0 PL=0
MOVL C00473 V=800.0 PL=0
MOVL C00474 V=800.0 PL=0
MOVL C00475 V=800.0 PL=0
MOVL C00476 V=800.0 PL=0
MOVL C00477 V=800.0 PL=0
MOVL C00478 V=800.0 PL=0
MOVL C00479 V=800.0 PL=0
MOVL C00480 V=800.0 PL=0
MOVL C00481 V=800.0 PL=0
MOVL C00482 V=800.0 PL=0
MOVL C00483 V=800.0 PL=0
MOVL C00484 V=800.0 PL=0
MOVL C00485 V=800.0 PL=0
MOVL C00486 V=800.0 PL=0
MOVL C00487 V=800.0 PL=0
MOVL C00488 V=800.0 PL=0
MOVL C00489 V=800.0 PL=0
MOVL C00490 V=800.0 PL=0
MOVL C00491 V=800.0 PL=0
MOVL C00492 V=800.0 PL=0
MOVL C00493 V=800.0 PL=0
MOVL C00494 V=800.0 PL=0
MOVL C00495 V=800.0 PL=0
MOVL C00496 V=800.0 PL=0
MOVL C00497 V=800.0 PL=0
MOVL C00498 V=800.0 PL=0
MOVL C00499 V=800.0 PL=0
MOVL C00500 V=800.0 PL=0
MOVL C00501 V=800.0 PL=0
MOVL C00502 V=800.0 PL=0
MOVL C00503 V=800.0 PL=0
MOVL C00504 V=800.0 PL=0
MOVL C00505 V=800.0 PL=0
MOVL C00506 V=800.0 PL=0
MOVL C00507 V=800.0 PL=0
MOVL C00508 V=800.0 PL=0
MOVL C00509 V=800.0 PL=0
MOVL C00510 V=800.0 PL=0
MOVL C00511 V=800.0 PL=0
MOVL C00512 V=800.0 PL=0
MOVL C00513 V=800.0 PL=0
MOVL C00514 V=800.0 PL=0
MOVL C00515 V=800.0 PL=0
MOVL C00516 V=800.0 PL=0
MOVL C00517 V=800.0 PL=0
MOVL C00518 V=800.0 PL=0
MOVL C00519 V=800.0 PL=0
MOVL C00520 V=800.0 PL=0
MOVL C00521 V=800.0 PL=0
MOVL C00522 V=800.0 PL=0
MOVL C00523 V=800.0 PL=0
MOVL C00524 V=800.0 PL=0
MOVL C00525 V=800.0 PL=0
MOVL C00526 V=800.0 PL=0
MOVL C00527 V=800.0 PL=0
MOVL C00528 V=800.0 PL=0
MOVL C00529 V=800.0 PL=0
MOVL C00530 V=800.0 PL=0
MOVL C00531 V=800.0 PL=0
MOVL C00532 V=800.0 PL=0
MOVL C00533 V=800.0 PL=0
MOVL C00534 V=800.0 PL=0
MOVL C00535 V=800.0 PL=0
MOVL C00536 V=800.0 PL=0
MOVL C00537 V=800.0 PL=0
MOVL C00538 V=800.0 PL=0
MOVL C00539 V=800.0 PL=0
MOVL C00540 V=800.0 PL=0
MOVL C00541 V=800.0 PL=0
MOVL C00542 V=800.0 PL=0
MOVL C00543 V=800.0 PL=0
MOVL C00544 V=800.0 PL=0
MOVL C00545 V=800.0 PL=0
MOVL C00546 V=800.0 PL=0
MOVL C00547 V=800.0 PL=0
MOVL C00548 V=800.0 PL=0
MOVL C00549 V=800.0 PL=0
MOVL C00550 V=800.0 PL=0
MOVL C00551 V=800.0 PL=0
MOVL C00552 V=800.0 PL=0
MOVL C00553 V=800.0 PL=0
MOVL C00554 V=800.0 PL=0
MOVL C00555 V=800.0 PL=0
MOVL C00556 V=800.0 PL=0
MOVL C00557 V=800.0 PL=0
MOVL C00558 V=800.0 PL=0
MOVL C00559 V=800.0 PL=0
MOVL C00560 V=800.0 PL=0
MOVL C00561 V=800.0 PL=0
MOVL C00562 V=800.0 PL=0
MOVL C00563 V=800.0 PL=0
MOVL C00564 V=800.0 PL=0
MOVL C00565 V=800.0 PL=0
MOVL C00566 V=800.0 PL=0
MOVL C00567 V=800.0 PL=0
MOVL C00568 V=800.0 PL=0
MOVL C00569 V=800.0 PL=0
MOVL C00570 V=800.0 PL=0
MOVL C00571 V=800.0 PL=0
MOVL C00572 V=800.0 PL=0
MOVL C00573 V=800.0 PL=0
MOVL C00574 V=800.0 PL=0
MOVL C00575 V=800.0 PL=0
MOVL C00576 V=800.0 PL=0
MOVL C00577 V=800.0 PL=0
MOVL C00578 V=800.0 PL=0
MOVL C00579 V=800.0 PL=0
MOVL C00580 V=800.0 PL=0
MOVL C00581 V=800.0 PL=0
MOVL C00582 V=800.0 PL=0
MOVL C00583 V=800.0 PL=0
MOVL C00584 V=800.0 PL=0
MOVL C00585 V=800.0 PL=0
MOVL C00586 V=800.0 PL=0
MOVL C00587 V=800.0 PL=0
MOVL C00588 V=800.0 PL=0
MOVL C00589 V=800.0 PL=0
MOVL C00590 V=800.0 PL=0
MOVL C00591 V=800.0 PL=0
MOVL C00592 V=800.0 PL=0
MOVL C00593 V=800.0 PL=0
MOVL C00594 V=800.0 PL=0
MOVL C00595 V=800.0 PL=0
MOVL C00596 V=800.0 PL=0
MOVL C00597 V=800.0 PL=0
MOVL C00598 V=800.0 PL=0
MOVL C00599 V=800.0 PL=0
MOVL C00600 V=800.0 PL=0
MOVL C00601 V=800.0 PL=0
MOVL C00602 V=800.0 PL=0
MOVL C00603 V=800.0 PL=0
MOVL C00604 V=800.0 PL=0
MOVL C00605 V=800.0 PL=0
MOVL C00606 V=800.0 PL=0
MOVL C00607 V=800.0 PL=0
MOVL C00608 V=800.0 PL=0
MOVL C00609 V=800.0 PL=0
MOVL C00610 V=800.0 PL=0
MOVL C00611 V=800.0 PL=0
MOVL C00612 V=800.0 PL=0
MOVL C00613 V=800.0 PL=0
MOVL C00614 V=800.0 PL=0
MOVL C00615 V=800.0 PL=0
MOVL C00616 V=800.0 PL=0
MOVL C00617 V=800.0 PL=0
MOVL C00618 V=800.0 PL=0
MOVL C00619 V=800.0 PL=0
MOVL C00620 V=800.0 PL=0
MOVL C00621 V=800.0 PL=0
MOVL C00622 V=800.0 PL=0
MOVL C00623 V=800.0 PL=0
MOVL C00624 V=800.0 PL=0
MOVL C00625 V=800.0 PL=0
MOVL C00626 V=800.0 PL=0
MOVL C00627 V=800.0 PL=0
MOVL C00628 V=800.0 PL=0
MOVL C00629 V=800.0 PL=0
MOVL C00630 V=800.0 PL=0
MOVL C00631 V=800.0 PL=0
MOVL C00632 V=800.0 PL=0
MOVL C00633 V=800.0 PL=0
MOVL C00634 V=800.0 PL=0
MOVL C00635 V=800.0 PL=0
MOVL C00636 V=800.0 PL=0
MOVL C00637 V=800.0 PL=0
MOVL C00638 V=800.0 PL=0
MOVL C00639 V=800.0 PL=0
MOVL C00640 V=800.0 PL=0
MOVL C00641 V=800.0 PL=0
MOVL C00642 V=800.0 PL=0
MOVL C00643 V=800.0 PL=0
MOVL C00644 V=800.0 PL=0
MOVL C00645 V=800.0 PL=0
MOVL C00646 V=800.0 PL=0
MOVL C00647 V=800.0 PL=0
MOVL C00648 V=800.0 PL=0
MOVL C00649 V=800.0 PL=0
MOVL C00650 V=800.0 PL=0
MOVL C00651 V=800.0 PL=0
MOVL C00652 V=800.0 PL=0
MOVL C00653 V=800.0 PL=0
MOVL C00654 V=800.0 PL=0
MOVL C00655 V=800.0 PL=0
MOVL C00656 V=800.0 PL=0
MOVL C00657 V=800.0 PL=0
MOVL C00658 V=800.0 PL=0
MOVL C00659 V=800.0 PL=0
MOVL C00660 V=800.0 PL=0
MOVL C00661 V=800.0 PL=0
MOVL C00662 V=800.0 PL=0
MOVL C00663 V=800.0 PL=0
MOVL C00664 V=800.0 PL=0
MOVL C00665 V=800.0 PL=0
MOVL C00666 V=800.0 PL=0
MOVL C00667 V=800.0 PL=0
MOVL C00668 V=800.0 PL=0
MOVL C00669 V=800.0 PL=0
MOVL C00670 V=800.0 PL=0
MOVL C00671 V=800.0 PL=0
MOVL C00672 V=800.0 PL=0
MOVL C00673 V=800.0 PL=0
MOVL C00674 V=800.0 PL=0
MOVL C00675 V=800.0 PL=0
MOVL C00676 V=800.0 PL=0
MOVL C00677 V=800.0 PL=0
MOVL C00678 V=800.0 PL=0
MOVL C00679 V=800.0 PL=0
MOVL C00680 V=800.0 PL=0
MOVL C00681 V=800.0 PL=0
MOVL C00682 V=800.0 PL=0
MOVL C00683 V=800.0 PL=0
MOVL C00684 V=800.0 PL=0
MOVL C00685 V=800.0 PL=0
MOVL C00686 V=800.0 PL=0
MOVL C00687 V=800.0 PL=0
MOVL C00688 V=800.0 PL=0
MOVL C00689 V=800.0 PL=0
MOVL C00690 V=800.0 PL=0
MOVL C00691 V=800.0 PL=0
MOVL C00692 V=800.0 PL=0
MOVL C00693 V=800.0 PL=0
MOVL C00694 V=800.0 PL=0
MOVL C00695 V=800.0 PL=0
MOVL C00696 V=800.0 PL=0
MOVL C00697 V=800.0 PL=0
MOVL C00698 V=800.0 PL=0
MOVL C00699 V=800.0 PL=0
MOVL C00700 V=800.0 PL=0
MOVL C00701 V=800.0 PL=0
MOVL C00702 V=800.0 PL=0
MOVL C00703 V=800.0 PL=0
MOVL C00704 V=800.0 PL=0
MOVL C00705 V=800.0 PL=0
MOVL C00706 V=800.0 PL=0
MOVL C00707 V=800.0 PL=0
MOVL C00708 V=800.0 PL=0
MOVL C00709 V=800.0 PL=0
MOVL C00710 V=800.0 PL=0
MOVL C00711 V=800.0 PL=0
MOVL C00712 V=800.0 PL=0
MOVL C00713 V=800.0 PL=0
MOVL C00714 V=800.0 PL=0
MOVL C00715 V=800.0 PL=0
MOVL C00716 V=800.0 PL=0
MOVL C00717 V=800.0 PL=0
MOVL C00718 V=800.0 PL=0
MOVL C00719 V=800.0 PL=0
MOVL C00720 V=800.0 PL=0
MOVL C00721 V=800.0 PL=0
MOVL C00722 V=800.0 PL=0
MOVL C00723 V=800.0 PL=0
MOVL C00724 V=800.0 PL=0
MOVL C00725 V=800.0 PL=0
MOVL C00726 V=800.0 PL=0
MOVL C00727 V=800.0 PL=0
MOVL C00728 V=800.0 PL=0
MOVL C00729 V=800.0 PL=0
MOVL C00730 V=800.0 PL=0
MOVL C00731 V=800.0 PL=0
MOVL C00732 V=800.0 PL=0
MOVL C00733 V=800.0 PL=0
MOVL C00734 V=800.0 PL=0
MOVL C00735 V=800.0 PL=0
MOVL C00736 V=800.0 PL=0
MOVL C00737 V=800.0 PL=0
MOVL C00738 V=800.0 PL=0
MOVL C00739 V=800.0 PL=0
MOVL C00740 V=800.0 PL=0
MOVL C00741 V=800.0 PL=0
MOVL C00742 V=800.0 PL=0
MOVL C00743 V=800.0 PL=0
MOVL C00744 V=800.0 PL=0
MOVL C00745 V=800.0 PL=0
MOVL C00746 V=800.0 PL=0
MOVL C00747 V=800.0 PL=0
MOVL C00748 V=800.0 PL=0
MOVL C00749 V=800.0 PL=0
MOVL C00750 V=800.0 PL=0
MOVL C00751 V=800.0 PL=0
MOVL C00752 V=800.0 PL=0
MOVL C00753 V=800.0 PL=0
MOVL C00754 V=800.0 PL=0
MOVL C00755 V=800.0 PL=0
MOVL C00756 V=800.0 PL=0
MOVL C00757 V=800.0 PL=0
MOVL C00758 V=800.0 PL=0
MOVL C00759 V=800.0 PL=0
MOVL C00760 V=800.0 PL=0
MOVL C00761 V=800.0 PL=0
MOVL C00762 V=800.0 PL=0
MOVL C00763 V=800.0 PL=0
MOVL C00764 V=800.0 PL=0
MOVL C00765 V=800.0 PL=0
MOVL C00766 V=800.0 PL=0
MOVL C00767 V=800.0 PL=0
MOVL C00768 V=800.0 PL=0
MOVL C00769 V=800.0 PL=0
MOVL C00770 V=800.0 PL=0
MOVL C00771 V=800.0 PL=0
MOVL C00772 V=800.0 PL=0
MOVL C00773 V=800.0 PL=0
MOVL C00774 V=800.0 PL=0
MOVL C00775 V=800.0 PL=0
MOVL C00776 V=800.0 PL=0
MOVL C00777 V=800.0 PL=0
MOVL C00778 V=800.0 PL=0
MOVL C00779 V=800.0 PL=0
MOVL C00780 V=800.0 PL=0
MOVL C00781 V=800.0 PL=0
MOVL C00782 V=800.0 PL=0
MOVL C00783 V=800.0 PL=0
MOVL C00784 V=800.0 PL=0
MOVL C00785 V=800.0 PL=0
MOVL C00786 V=800.0 PL=0
MOVL C00787 V=800.0 PL=0
MOVL C00788 V=800.0 PL=0
MOVL C00789 V=800.0 PL=0
MOVL C00790 V=800.0 PL=0
MOVL C00791 V=800.0 PL=0
MOVL C00792 V=800.0 PL=0
MOVL C00793 V=800.0 PL=0
MOVL C00794 V=800.0 PL=0
MOVL C00795 V=800.0 PL=0
MOVL C00796 V=800.0 PL=0
MOVL C00797 V=800.0 PL=0
MOVL C00798 V=800.0 PL=0
MOVL C00799 V=800.0 PL=0
MOVL C00800 V=800.0 PL=0
MOVL C00801 V=800.0 PL=0
MOVL C00802 V=800.0 PL=0
MOVL C00803 V=800.0 PL=0
MOVL C00804 V=800.0 PL=0
MOVL C00805 V=800.0 PL=0
MOVL C00806 V=800.0 PL=0
MOVL C00807 V=800.0 PL=0
MOVL C00808 V=800.0 PL=0
MOVL C00809 V=800.0 PL=0
MOVL C00810 V=800.0 PL=0
MOVL C00811 V=800.0 PL=0
MOVL C00812 V=800.0 PL=0
MOVL C00813 V=800.0 PL=0
MOVL C00814 V=800.0 PL=0
MOVL C00815 V=800.0 PL=0
MOVL C00816 V=800.0 PL=0
MOVL C00817 V=800.0 PL=0
MOVL C00818 V=800.0 PL=0
MOVL C00819 V=800.0 PL=0
MOVL C00820 V=800.0 PL=0
MOVL C00821 V=800.0 PL=0
MOVL C00822 V=800.0 PL=0
MOVL C00823 V=800.0 PL=0
MOVL C00824 V=800.0 PL=0
MOVL C00825 V=800.0 PL=0
MOVL C00826 V=800.0 PL=0
MOVL C00827 V=800.0 PL=0
MOVL C00828 V=800.0 PL=0
MOVL C00829 V=800.0 PL=0
MOVL C00830 V=800.0 PL=0
MOVL C00831 V=800.0 PL=0
MOVL C00832 V=800.0 PL=0
MOVL C00833 V=800.0 PL=0
MOVL C00834 V=800.0 PL=0
MOVL C00835 V=800.0 PL=0
MOVL C00836 V=800.0 PL=0
MOVL C00837 V=800.0 PL=0
MOVL C00838 V=800.0 PL=0
MOVL C00839 V=800.0 PL=0
MOVL C00840 V=800.0 PL=0
MOVL C00841 V=800.0 PL=0
MOVL C00842 V=800.0 PL=0
MOVL C00843 V=800.0 PL=0
MOVL C00844 V=800.0 PL=0
MOVL C00845 V=800.0 PL=0
MOVL C00846 V=800.0 PL=0
MOVL C00847 V=800.0 PL=0
MOVL C00848 V=800.0 PL=0
MOVL C00849 V=800.0 PL=0
MOVL C00850 V=800.0 PL=0
MOVL C00851 V=800.0 PL=0
MOVL C00852 V=800.0 PL=0
MOVL C00853 V=800.0 PL=0
MOVL C00854 V=800.0 PL=0
MOVL C00855 V=800.0 PL=0
MOVL C00856 V=800.0 PL=0
MOVL C00857 V=800.0 PL=0
MOVL C00858 V=800.0 PL=0
MOVL C00859 V=800.0 PL=0
MOVL C00860 V=800.0 PL=0
MOVL C00861 V=800.0 PL=0
MOVL C00862 V=800.0 PL=0
MOVL C00863 V=800.0 PL=0
MOVL C00864 V=800.0 PL=0
MOVL C00865 V=800.0 PL=0
MOVL C00866 V=800.0 PL=0
MOVL C00867 V=800.0 PL=0
MOVL C00868 V=800.0 PL=0
MOVL C00869 V=800.0 PL=0
MOVL C00870 V=800.0 PL=0
MOVL C00871 V=800.0 PL=0
MOVL C00872 V=800.0 PL=0
MOVL C00873 V=800.0 PL=0
MOVL C00874 V=800.0 PL=0
MOVL C00875 V=800.0 PL=0
MOVL C00876 V=800.0 PL=0
MOVL C00877 V=800.0 PL=0
MOVL C00878 V=800.0 PL=0
MOVL C00879 V=800.0 PL=0
MOVL C00880 V=800.0 PL=0
MOVL C00881 V=800.0 PL=0
MOVL C00882 V=800.0 PL=0
MOVL C00883 V=800.0 PL=0
MOVL C00884 V=800.0 PL=0
MOVL C00885 V=800.0 PL=0
MOVL C00886 V=800.0 PL=0
MOVL C00887 V=800.0 PL=0
MOVL C00888 V=800.0 PL=0
MOVL C00889 V=800.0 PL=0
MOVL C00890 V=800.0 PL=0
MOVL C00891 V=800.0 PL=0
MOVL C00892 V=800.0 PL=0
MOVL C00893 V=800.0 PL=0
MOVL C00894 V=800.0 PL=0
MOVL C00895 V=800.0 PL=0
MOVL C00896 V=800.0 PL=0
MOVL C00897 V=800.0 PL=0
MOVL C00898 V=800.0 PL=0
MOVL C00899 V=800.0 PL=0
MOVL C00900 V=800.0 PL=0
MOVL C00901 V=800.0 PL=0
MOVL C00902 V=800.0 PL=0
MOVL C00903 V=800.0 PL=0
MOVL C00904 V=800.0 PL=0
MOVL C00905 V=800.0 PL=0
MOVL C00906 V=800.0 PL=0
MOVL C00907 V=800.0 PL=0
MOVL C00908 V=800.0 PL=0
MOVL C00909 V=800.0 PL=0
MOVL C00910 V=800.0 PL=0
MOVL C00911 V=800.0 PL=0
MOVL C00912 V=800.0 PL=0
MOVL C00913 V=800.0 PL=0
MOVL C00914 V=800.0 PL=0
MOVL C00915 V=800.0 PL=0
MOVL C00916 V=800.0 PL=0
MOVL C00917 V=800.0 PL=0
MOVL C00918 V=800.0 PL=0
MOVL C00919 V=800.0 PL=0
MOVL C00920 V=800.0 PL=0
MOVL C00921 V=800.0 PL=0
MOVL C00922 V=800.0 PL=0
MOVL C00923 V=800.0 PL=0
MOVL C00924 V=800.0 PL=0
MOVL C00925 V=800.0 PL=0
MOVL C00926 V=800.0 PL=0
MOVL C00927 V=800.0 PL=0
MOVL C00928 V=800.0 PL=0
MOVL C00929 V=800.0 PL=0
MOVL C00930 V=800.0 PL=0
MOVL C00931 V=800.0 PL=0
MOVL C00932 V=800.0 PL=0
MOVL C00933 V=800.0 PL=0
MOVL C00934 V=800.0 PL=0
MOVL C00935 V=800.0 PL=0
MOVL C00936 V=800.0 PL=0
MOVL C00937 V=800.0 PL=0
MOVL C00938 V=800.0 PL=0
MOVL C00939 V=800.0 PL=0
MOVL C00940 V=800.0 PL=0
MOVL C00941 V=800.0 PL=0
MOVL C00942 V=800.0 PL=0
MOVL C00943 V=800.0 PL=0
MOVL C00944 V=800.0 PL=0
MOVL C00945 V=800.0 PL=0
MOVL C00946 V=800.0 PL=0
MOVL C00947 V=800.0 PL=0
MOVL C00948 V=800.0 PL=0
MOVL C00949 V=800.0 PL=0
MOVL C00950 V=800.0 PL=0
MOVL C00951 V=800.0 PL=0
MOVL C00952 V=800.0 PL=0
MOVL C00953 V=800.0 PL=0
MOVL C00954 V=800.0 PL=0
MOVL C00955 V=800.0 PL=0
MOVL C00956 V=800.0 PL=0
MOVL C00957 V=800.0 PL=0
MOVL C00958 V=800.0 PL=0
MOVL C00959 V=800.0 PL=0
MOVL C00960 V=800.0 PL=0
MOVL C00961 V=800.0 PL=0
MOVL C00962 V=800.0 PL=0
MOVL C00963 V=800.0 PL=0
MOVL C00964 V=800.0 PL=0
MOVL C00965 V=800.0 PL=0
MOVL C00966 V=800.0 PL=0
MOVL C00967 V=800.0 PL=0
MOVL C00968 V=800.0 PL=0
MOVL C00969 V=800.0 PL=0
MOVL C00970 V=800.0 PL=0
MOVL C00971 V=800.0 PL=0
MOVL C00972 V=800.0 PL=0
MOVL C00973 V=800.0 PL=0
MOVL C00974 V=800.0 PL=0
MOVL C00975 V=800.0 PL=0
MOVL C00976 V=800.0 PL=0
MOVL C00977 V=800.0 PL=0
MOVL C00978 V=800.0 PL=0
MOVL C00979 V=800.0 PL=0
MOVL C00980 V=800.0 PL=0
MOVL C00981 V=800.0 PL=0
MOVL C00982 V=800.0 PL=0
MOVL C00983 V=800.0 PL=0
MOVL C00984 V=800.0 PL=0
MOVL C00985 V=800.0 PL=0
MOVL C00986 V=800.0 PL=0
MOVL C00987 V=800.0 PL=0
MOVL C00988 V=800.0 PL=0
MOVL C00989 V=800.0 PL=0
MOVL C00990 V=800.0 PL=0
MOVL C00991 V=800.0 PL=0
MOVL C00992 V=800.0 PL=0
MOVL C00993 V=800.0 PL=0
MOVL C00994 V=800.0 PL=0
MOVL C00995 V=800.0 PL=0
MOVL C00996 V=800.0 PL=0
MOVL C00997 V=800.0 PL=0
MOVL C00998 V=800.0 PL=0
MOVL C00999 V=800.0 PL=0
MOVL C01000 V=800.0 PL=0
MOVL C01001 V=800.0 PL=0
MOVL C01002 V=800.0 PL=0
MOVL C01003 V=800.0 PL=0
MOVL C01004 V=800.0 PL=0
MOVL C01005 V=800.0 PL=0
MOVL C01006 V=800.0 PL=0
MOVL C01007 V=800.0 PL=0
MOVL C01008 V=800.0 PL=0
MOVL C01009 V=800.0 PL=0
MOVL C01010 V=800.0 PL=0
MOVL C01011 V=800.0 PL=0
MOVL C01012 V=800.0 PL=0
MOVL C01013 V=800.0 PL=0
MOVL C01014 V=800.0 PL=0
MOVL C01015 V=800.0 PL=0
MOVL C01016 V=800.0 PL=0
MOVL C01017 V=800.0 PL=0
MOVL C01018 V=800.0 PL=0
MOVL C01019 V=800.0 PL=0
MOVL C01020 V=800.0 PL=0
MOVL C01021 V=800.0 PL=0
MOVL C01022 V=800.0 PL=0
MOVL C01023 V=800.0 PL=0
MOVL C01024 V=800.0 PL=0
MOVL C01025 V=800.0 PL=0
MOVL C01026 V=800.0 PL=0
MOVL C01027 V=800.0 PL=0
MOVL C01028 V=800.0 PL=0
MOVL C01029 V=800.0 PL=0
MOVL C01030 V=800.0 PL=0
MOVL C01031 V=800.0 PL=0
MOVL C01032 V=800.0 PL=0
MOVL C01033 V=800.0 PL=0
MOVL C01034 V=800.0 PL=0
MOVL C01035 V=800.0 PL=0
MOVL C01036 V=800.0 PL=0
MOVL C01037 V=800.0 PL=0
MOVL C01038 V=800.0 PL=0
MOVL C01039 V=800.0 PL=0
MOVL C01040 V=800.0 PL=0
MOVL C01041 V=800.0 PL=0
MOVL C01042 V=800.0 PL=0
MOVL C01043 V=800.0 PL=0
MOVL C01044 V=800.0 PL=0
MOVL C01045 V=800.0 PL=0
MOVL C01046 V=800.0 PL=0
MOVL C01047 V=800.0 PL=0
MOVL C01048 V=800.0 PL=0
MOVL C01049 V=800.0 PL=0
MOVL C01050 V=800.0 PL=0
MOVL C01051 V=800.0 PL=0
MOVL C01052 V=800.0 PL=0
MOVL C01053 V=800.0 PL=0
MOVL C01054 V=800.0 PL=0
MOVL C01055 V=800.0 PL=0
